(* IEC 61131-3 sources: std_i2980_v2.06_cp053/Source/IMM/ieccontrol/GlobalBaseArchives (part 19) *)

(* ---- ABRegisterDelay.pu ---- *)
(*
@h    ! WARNING !
@h    The Kemro K2 system (including software) only meets category B according to EN 954-1,
@h    thus it is not intended for usage in safety-relevant control applications in the field
@h    of personal safety (e.g. emergency stop).
@h    To implement potentially necessary safety-relevant control tasks, always use additional
@h    external safety devices that are intended for the particular purpose, and meet the necessary
@h    functional safety.
@h    For further information see EN 954-1 (EN ISO 13849-1) and/or the K2-x00 user manual, chapter
@h    "CE conformity, directives and standards".

Delaytime generator for movement and deviceregistration.
*)

ALGORITHM_BLOCK ABRegisterDelay #DUMMY_EDIT_BLOCK

SYSTEM_VAR
 sv_iRegistrationCounter : DINT (* Registrationcounter for delaytime generation *);
END_VAR

(*
Returns a delaytime which is raised by 10ms every call.
*)

ALGORITHM aGet

VAR_OUTPUT
 Time : TIME;
END_VAR
#BEGIN_EDIT_BLOCK
(**************************************** WARNING ********************************************
 *** The KEBA Kemro K2 System including software is not intended for safety control tasks! ***
 ***                       For further information see Comment tab!                        ***
 *********************************************************************************************)

// increment Register counter
sv_iRegistrationCounter := sv_iRegistrationCounter + 1;
// calculate delaytime for registration
Time := T#10ms * sv_iRegistrationCounter;

;#END_EDIT_BLOCK END_ALGORITHM

(*
Resetting the delaytime to make it ready for another registration sequence.
*)

ALGORITHM aReset

#BEGIN_EDIT_BLOCK
(**************************************** WARNING ********************************************
 *** The KEBA Kemro K2 System including software is not intended for safety control tasks! ***
 ***                       For further information see Comment tab!                        ***
 *********************************************************************************************)

// reset devicesRegistered counter
sv_iRegistrationCounter := 0;

;#END_EDIT_BLOCK END_ALGORITHM

END_ALGORITHM_BLOCK

#END_OF_IEC_PART

@Puma @IecEditor 6 10 @Pou 25
@@@BEG_Comment@@@
@h    ! WARNING !
@h    The Kemro K2 system (including software) only meets category B according to EN 954-1,
@h    thus it is not intended for usage in safety-relevant control applications in the field
@h    of personal safety (e.g. emergency stop).
@h    To implement potentially necessary safety-relevant control tasks, always use additional
@h    external safety devices that are intended for the particular purpose, and meet the necessary
@h    functional safety.
@h    For further information see EN 954-1 (EN ISO 13849-1) and/or the K2-x00 user manual, chapter
@h    "CE conformity, directives and standards".

Delaytime generator for movement and deviceregistration.
@@@END_Comment@@@

@BEG_Contents

@BEG_Func
@RT(17)FuncTreeContainer
0
@END_Func

@BEG_Const
@RT(18)ConstTreeContainer
0
@END_Const

@BEG_Export

@BEG_Kind
@ALGORITHM_BLOCK @RT(15)ABRegisterDelay @STRUCTURED_TEXT
@RT(0) @RT(0) @RT(0)
@END_Kind

@BEG_Dcl
@RT(16)DclTreeContainer
1
@Var @RT(23)sv_iRegistrationCounter @RT(0) @T @F @DT @RT(4)DINT @RT(0) @T @T @BASIC 0 @F
@F @F
@T
@BEG_Attrib
3 @RT(0) @RT(44)Registrationcounter for delaytime generation @RT(0)
@END_Attrib
1 8 @F @F @F @F

@END_Dcl

@END_Export

@BEG_Body

2

@BEG_Export

@BEG_Algo
@ALGORITHM @RT(4)aGet @STRUCTURED_TEXT
@RT(0) @RT(0) @RT(0) @F @F
@END_Algo

@BEG_Dcl
@RT(16)DclTreeContainer
1
@Var @RT(4)Time @RT(0) @T @F @DT @RT(4)TIME @RT(0) @T @T @BASIC 0 @F
@F @F
@T
@BEG_Attrib
3 @RT(0) @RT(0) @RT(0)
@END_Attrib
1 3 @F @F @F @F

@END_Dcl

@END_Export

@BEG_Export

@BEG_Algo
@ALGORITHM @RT(6)aReset @STRUCTURED_TEXT
@RT(0) @RT(0) @RT(0) @F @F
@END_Algo

@BEG_Dcl
@RT(16)DclTreeContainer
0
@END_Dcl

@END_Export

@BEG_Body
@TL(10)
(**************************************** WARNING ********************************************
 *** The KEBA Kemro K2 System including software is not intended for safety control tasks! ***
 ***                       For further information see Comment tab!                        ***
 *********************************************************************************************)

// increment Register counter
sv_iRegistrationCounter := sv_iRegistrationCounter + 1;
// calculate delaytime for registration
Time := T#10ms * sv_iRegistrationCounter;

@END_Body

@@@BEG_Comment@@@
@TL(1)
Returns a delaytime which is raised by 10ms every call.
@@@END_Comment@@@

@BEG_Body
@TL(8)
(**************************************** WARNING ********************************************
 *** The KEBA Kemro K2 System including software is not intended for safety control tasks! ***
 ***                       For further information see Comment tab!                        ***
 *********************************************************************************************)

// reset devicesRegistered counter
sv_iRegistrationCounter := 0;

@END_Body

@@@BEG_Comment@@@
@TL(1)
Resetting the delaytime to make it ready for another registration sequence.
@@@END_Comment@@@
@END_Body

@END_Contents

(* ---- ABResourceLockManager.pu ---- *)
IMPORT_OVER_LISTFILE
 STOP_PROCESS_ALGORITHM
, tsResourceLock
, TON

END_IMPORT

ALGORITHM_BLOCK ABResourceLockManager #DUMMY_EDIT_BLOCK

SYSTEM_OBJECT
 PU_Task_7 : TASK;
 TaskSlow : TASK;
END_OBJECT

VAR
 mpResource : REFTO tsResourceLock;
 fbTimeout : TON;
 mbTimeoutUsed : BOOL;
 mName : STRING(31);
END_VAR

ALGORITHM aRequest

#BEGIN_EDIT_BLOCK

IF (mpResource^.iRequest <> 0) THEN // lock request
    IF (mpResource^.iLocked MOD 2 = 0) THEN  // is unlocked
        mpResource^.iResponse := mpResource^.iRequest;
        mpResource^.iLocked := mpResource^.iLocked + 1;  // do lock
        IF (mbTimeoutUsed) THEN
            fbTimeout(IN := FALSE);
            START_PROCESS_ALGORITHM(paTimeout);
        END_IF;
    END_IF;
END_IF;

;#END_EDIT_BLOCK END_ALGORITHM

POSTUPDATE_ALGORITHM pRequest ON PU_Task_7(1) WITH mpResource^.iRequest

#BEGIN_EDIT_BLOCK
aRequest();

;#END_EDIT_BLOCK END_ALGORITHM

POSTUPDATE_ALGORITHM pRelease ON PU_Task_7(2) WITH mpResource^.iResponse

#BEGIN_EDIT_BLOCK
IF (mpResource^.iResponse = 0) THEN
    IF ((mpResource^.iLocked MOD 2 = 1)) THEN // locked
        mpResource^.iLocked := mpResource^.iLocked + 1; // unlock
        mpResource^.iRequest := 0;
        IF (mbTimeoutUsed) THEN
            STOP_PROCESS_ALGORITHM(paTimeout);
        END_IF;
    END_IF;
END_IF;

;#END_EDIT_BLOCK END_ALGORITHM

ALGORITHM aInit

VAR_INPUT
 sName : STRING(31);
 pResource : REFTO tsResourceLock;
 dTimeout : TIME;
END_VAR
#BEGIN_EDIT_BLOCK
mpResource := pResource;
mbTimeoutUsed := dTimeout > T#0s;
fbTimeout.PT := dTimeout;
mName := sName;
aRequest();

;#END_EDIT_BLOCK END_ALGORITHM

PROCESS_ALGORITHM paTimeout ON TaskSlow

VAR
 dummy : DINT;
END_VAR
#BEGIN_EDIT_BLOCK
fbTimeout(IN := (mpResource^.iLocked MOD 2 = 1));
IF (fbTimeout.Q) THEN
    dummy := Print("ABResourceLockManager(%s): lock timeout for lockid 0x%08x", mName, mpResource^.iResponse);
    mpResource^.iResponse := 0;
END_IF;

;#END_EDIT_BLOCK END_ALGORITHM

END_ALGORITHM_BLOCK

#END_OF_IEC_PART

@Puma @IecEditor 6 159 @Pou 25
@@@BEG_Comment@@@

@@@END_Comment@@@

@BEG_Contents

@BEG_Func
@RT(17)FuncTreeContainer
1
@Var @RT(22)STOP_PROCESS_ALGORITHM @RT(0) @T @T @DERIVED 0 @F @RT(23)KEBA_STANDARD_PROCEDURE @F
@T
@BEG_Attrib
0 @RT(0) @RT(0)
@END_Attrib
1 1 @F @F @F @F

@END_Func

@BEG_Const
@RT(18)ConstTreeContainer
0
@END_Const

@BEG_Export

@BEG_Kind
@ALGORITHM_BLOCK @RT(21)ABResourceLockManager @STRUCTURED_TEXT
@RT(0) @RT(0) @RT(0)
@END_Kind

@BEG_Dcl
@RT(16)DclTreeContainer
6
@Var @RT(9)PU_Task_7 @RT(0) @T @T @RENAMED 0 @T @T @DT @RT(4)TASK @RT(0) @T @T @BASIC 0 @F
@F @F
@T
@BEG_Attrib
3 @RT(0) @RT(0) @RT(0)
@END_Attrib
1 7 @F @F @F @F

@Var @RT(10)mpResource @RT(0) @T @T @REFTO 0 @F @DERIVED 0 @T @T @DT @RT(14)tsResourceLock @RT(0) @T @T @UNKNOWN 0 @F
@F @F
@T
@BEG_Attrib
3 @RT(0) @RT(0) @RT(0)
@END_Attrib
1 0 @F @F @F @F

@Var @RT(8)TaskSlow @RT(0) @T @T @RENAMED 0 @T @T @DT @RT(4)TASK @RT(0) @T @T @BASIC 0 @F
@F @F
@T
@BEG_Attrib
3 @RT(0) @RT(0) @RT(0)
@END_Attrib
1 7 @F @F @F @F

@Var @RT(9)fbTimeout @RT(0) @T @T @DERIVED 0 @T @T @DT @RT(3)TON @RT(0) @T @T @UNKNOWN 0 @F
@F @F
@T
@BEG_Attrib
3 @RT(0) @RT(0) @RT(0)
@END_Attrib
1 0 @F @F @F @F

@Var @RT(13)mbTimeoutUsed @RT(0) @T @F @DT @RT(4)BOOL @RT(0) @T @T @BASIC 0 @F
@F @F
@T
@BEG_Attrib
3 @RT(0) @RT(0) @RT(0)
@END_Attrib
1 0 @F @F @F @F

@Var @RT(5)mName @RT(0) @T @F @DT @RT(10)STRING(31) @RT(0) @T @T @STRING 0 @F @RT(2)31 @F
@F @F
@T
@BEG_Attrib
3 @RT(0) @RT(0) @RT(0)
@END_Attrib
1 0 @F @F @F @F

@END_Dcl

@END_Export

@BEG_Body

5

@BEG_Export

@BEG_Algo
@ALGORITHM @RT(8)aRequest @STRUCTURED_TEXT
@RT(0) @RT(0) @RT(0) @F @F
@END_Algo

@BEG_Dcl
@RT(16)DclTreeContainer
0
@END_Dcl

@END_Export

@BEG_Export

@BEG_Algo
@POSTUPDATE_ALGORITHM @RT(8)pRequest @STRUCTURED_TEXT
@RT(0) @RT(20)mpResource^.iRequest @RT(12)PU_Task_7(1) @F @F
@END_Algo

@BEG_Dcl
@RT(16)DclTreeContainer
0
@END_Dcl

@END_Export

@BEG_Export

@BEG_Algo
@POSTUPDATE_ALGORITHM @RT(8)pRelease @STRUCTURED_TEXT
@RT(0) @RT(21)mpResource^.iResponse @RT(12)PU_Task_7(2) @F @F
@END_Algo

@BEG_Dcl
@RT(16)DclTreeContainer
0
@END_Dcl

@END_Export

@BEG_Export

@BEG_Algo
@ALGORITHM @RT(5)aInit @STRUCTURED_TEXT
@RT(0) @RT(0) @RT(0) @F @F
@END_Algo

@BEG_Dcl
@RT(16)DclTreeContainer
3
@Var @RT(5)sName @RT(0) @T @F @DT @RT(10)STRING(31) @RT(0) @T @T @STRING 0 @F @RT(2)31 @F
@F @F
@T
@BEG_Attrib
3 @RT(0) @RT(0) @RT(0)
@END_Attrib
1 1 @F @F @F @F

@Var @RT(9)pResource @RT(0) @T @T @REFTO 0 @F @DERIVED 0 @T @T @DT @RT(14)tsResourceLock @RT(0) @T @T @UNKNOWN 0 @F
@F @F
@T
@BEG_Attrib
3 @RT(0) @RT(0) @RT(0)
@END_Attrib
1 1 @F @F @F @F

@Var @RT(8)dTimeout @RT(0) @T @F @DT @RT(4)TIME @RT(0) @T @T @BASIC 0 @F
@F @F
@T
@BEG_Attrib
3 @RT(0) @RT(0) @RT(0)
@END_Attrib
1 1 @F @F @F @F

@END_Dcl

@END_Export

@BEG_Export

@BEG_Algo
@PROCESS_ALGORITHM @RT(9)paTimeout @STRUCTURED_TEXT
@RT(0) @RT(0) @RT(8)TaskSlow @F @F
@END_Algo

@BEG_Dcl
@RT(16)DclTreeContainer
1
@Var @RT(5)dummy @RT(0) @T @F @DT @RT(4)DINT @RT(0) @T @T @BASIC 0 @F
@F @F
@T
@BEG_Attrib
3 @RT(0) @RT(0) @RT(0)
@END_Attrib
1 0 @F @F @F @F

@END_Dcl

@END_Export

@BEG_Body
@TL(12)

IF (mpResource^.iRequest <> 0) THEN // lock request
    IF (mpResource^.iLocked MOD 2 = 0) THEN  // is unlocked
        mpResource^.iResponse := mpResource^.iRequest;
        mpResource^.iLocked := mpResource^.iLocked + 1;  // do lock
        IF (mbTimeoutUsed) THEN
            fbTimeout(IN := FALSE);
            START_PROCESS_ALGORITHM(paTimeout);
        END_IF;
    END_IF;
END_IF;

@END_Body

@@@BEG_Comment@@@
@TL(0)

@@@END_Comment@@@

@BEG_Body
@TL(2)
aRequest();

@END_Body

@@@BEG_Comment@@@
@TL(0)

@@@END_Comment@@@

@BEG_Body
@TL(10)
IF (mpResource^.iResponse = 0) THEN
    IF ((mpResource^.iLocked MOD 2 = 1)) THEN // locked
        mpResource^.iLocked := mpResource^.iLocked + 1; // unlock
        mpResource^.iRequest := 0;
        IF (mbTimeoutUsed) THEN
            STOP_PROCESS_ALGORITHM(paTimeout);
        END_IF;
    END_IF;
END_IF;

@END_Body

@@@BEG_Comment@@@
@TL(0)

@@@END_Comment@@@

@BEG_Body
@TL(6)
mpResource := pResource;
mbTimeoutUsed := dTimeout > T#0s;
fbTimeout.PT := dTimeout;
mName := sName;
aRequest();

@END_Body

@@@BEG_Comment@@@
@TL(0)

@@@END_Comment@@@

@BEG_Body
@TL(6)
fbTimeout(IN := (mpResource^.iLocked MOD 2 = 1));
IF (fbTimeout.Q) THEN
    dummy := Print("ABResourceLockManager(%s): lock timeout for lockid 0x%08x", mName, mpResource^.iResponse);
    mpResource^.iResponse := 0;
END_IF;

@END_Body

@@@BEG_Comment@@@
@TL(0)

@@@END_Comment@@@
@END_Body

@END_Contents

(* ---- ABStepOutput.pu ---- *)
(*
@h    ! WARNING !
@h    The Kemro K2 system (including software) only meets category B according to EN 954-1,
@h    thus it is not intended for usage in safety-relevant control applications in the field
@h    of personal safety (e.g. emergency stop).
@h    To implement potentially necessary safety-relevant control tasks, always use additional
@h    external safety devices that are intended for the particular purpose, and meet the necessary
@h    functional safety.
@h    For further information see EN 954-1 (EN ISO 13849-1) and/or the K2-x00 user manual, chapter
@h    "CE conformity, directives and standards".

Do step with low and high output value.
*)

IMPORT_OVER_LISTFILE
 GET_TASK_INTERVAL
, cApplPlasticsNoError
, ABConstMovement
, tsVelPre
, tMoveIdent
, R_TRIG

END_IMPORT

ALGORITHM_BLOCK ABStepOutput #DUMMY_EDIT_BLOCK

VAR
 abConstMovement : ABConstMovement;
 CycleTime : TIME (* (of capturing) *);
 bStarted : BOOL;
 mpConstant : REFTO tsVelPre;
 mprMaxSpeed : REFTO REAL;
END_VAR

ALGORITHM aInit

VAR_INPUT
 pConst : REFTO tsVelPre (* pointer to systemvariable that contains profile *);
 MoveId : tMoveIdent (* moveId of constant movement *);
 prMaxSpeed : REFTO REAL;
END_VAR
#BEGIN_EDIT_BLOCK
(**************************************** WARNING ********************************************
 *** The KEBA Kemro K2 System including software is not intended for safety control tasks! ***
 ***                       For further information see Comment tab!                        ***
 *********************************************************************************************)

mpConstant := pConst;

abConstMovement.aInit(pConst := pConst,
                      MoveId := MoveId);

mprMaxSpeed := prMaxSpeed;

;#END_EDIT_BLOCK END_ALGORITHM

(*
Output profile for back pressure calibration
and measure the pressure input
*)

ALGORITHM aRun

VAR_INPUT
 bStart : BOOL (* start constant calib block *);
 bStop : BOOL (* stop constant calib block *);
 bDirection : BOOL (* movement direction *);
 rActPos : REAL (* actual position *);
 rTargetPos : REAL (* target position *);
 bUsePosDetect : BOOL (* TRUE: movement should stop at target position *);
 dDelayTimeOn : TIME (* Delay Time between preoutput and  constoutput *);
 dDelayTimeOff : TIME (* Delay Time between pump stop and bActive FALSE *);
 rPositionUp : REAL;
 rPositionDown : REAL;
 rLowOutput : REAL;
 rHighOutput : REAL;
 dMaxMoveTime : TIME;
 rStopRamp : REAL;
END_VAR

VAR_OUTPUT
 bActive : BOOL (* movement is active *);
 rOutputPre : REAL (* pressure output *);
 rOutputVel : REAL (* velocity output *);
 bPreOutputReached : BOOL (* preoutput ready *);
 bError : BOOL (* flag to indicate if error occured *);
 iErrorInfo : DINT (* additional error info *);
END_VAR

VAR
 fbREdge_Start : R_TRIG;
 iStage : DINT;
 bUeStopRamp : BOOL;
 rSavePreOutput : REAL;
 rSaveRamp : REAL;
 rDownPosition : REAL;
 rUpPosition : REAL;
 dMinDelayTimStop : TIME := T#50ms;
END_VAR
#BEGIN_EDIT_BLOCK
(**************************************** WARNING ********************************************
 *** The KEBA Kemro K2 System including software is not intended for safety control tasks! ***
 ***                       For further information see Comment tab!                        ***
 *********************************************************************************************)

fbREdge_Start(CLK := bStart);
IF fbREdge_Start.Q THEN
   iStage := 1;
   bStarted := TRUE;

   rDownPosition := rPositionDown;
   rUpPosition := rPositionUp;

   rSavePreOutput := mpConstant^.Velocity.PreOutput.rOutputValue;
   mpConstant^.Velocity.PreOutput.rOutputValue :=  rHighOutput;
   mpConstant^.Velocity.PreOutput.rRamp := 1.0e10;
   rSaveRamp := mpConstant^.Velocity.Output.rRamp;

   IF (rStopRamp > 0.0) THEN
      bUeStopRamp := TRUE;
      mpConstant^.Velocity.Output.rRamp := rStopRamp;
   ELSE
      bUeStopRamp := FALSE;
   END_IF;

   abConstMovement.aRun(bStart := FALSE);
   CycleTime := GET_TASK_INTERVAL();
END_IF;
IF bStop THEN
    bStarted := FALSE;
END_IF;

IF bStarted THEN
   //call const movement block
   abConstMovement.aRun(bStart := bStart,
                        bStop := bStop,
                        bDirection := bDirection,
                        rActPos := rActPos,
                        rTargetPos := rTargetPos,
                        bUsePosDetect := bUsePosDetect,
                        rStartOutputPre := 0.0,
                        rStartOutputVel := rHighOutput,
                        dDelayTimeOn := dDelayTimeOn,
                        dDelayTimeOff := MAX(dDelayTimeOff, dMinDelayTimStop),
                        dMaxTime := dMaxMoveTime);

   IF (bDirection AND (rActPos >=  rDownPosition)) OR
      (NOT bDirection AND (rActPos <=  rDownPosition)) THEN
      iStage := 3;
   ELSIF (bDirection AND (rActPos >=  rUpPosition) ) OR
      (NOT bDirection AND (rActPos <=  rUpPosition)) THEN
      iStage := 2;
   END_IF;

   (* to do a jump without a ramp we directly output the low value *)
   IF iStage = 1 THEN
      rOutputVel := MIN(rLowOutput,mpConstant^.Velocity.Output.rOutputValue);
   ELSIF iStage = 2 THEN
      IF (bUeStopRamp) THEN
         rOutputVel := MIN(abConstMovement.aRun.rOutputVel, rHighOutput);
      ELSE
         rOutputVel := rHighOutput;
      END_IF;
   ELSIF iStage = 3 THEN
      IF (bUeStopRamp) THEN
         rOutputVel := abConstMovement.aRun.rOutputVel;
      ELSE
         rOutputVel := MIN(rLowOutput, abConstMovement.aRun.rOutputVel);
      END_IF;
   ELSE
      rOutputVel := 0.0;
   END_IF;

   rOutputPre := abConstMovement.aRun.rOutputPre;
   IF (bDirection AND (rActPos <  rTargetPos)) OR
      (NOT bDirection AND (rActPos >  rTargetPos)) THEN
      bActive := TRUE;
      bPreOutputReached := TRUE;
   ELSE
      bActive := abConstMovement.aRun.bActive;
      bPreOutputReached := abConstMovement.aRun.bPreOutputReached;
   END_IF;

   bError := abConstMovement.aRun.bError;
ELSE
   // not started
   rOutputPre := 0.0;
   rOutputVel := 0.0;
   bPreOutputReached := TRUE;
   bActive := FALSE;
   bError := FALSE;

   abConstMovement.aRun(bStart := FALSE,
                        bStop := TRUE);
END_IF;

//finished ramping down -> switch off
IF bStarted AND NOT abConstMovement.aRun.bActive THEN
   bStarted := FALSE;
   rOutputPre := 0.0;
   rOutputVel := 0.0;
   mpConstant^.Velocity.PreOutput.rOutputValue := rSavePreOutput;
   mpConstant^.Velocity.Output.rRamp := rSaveRamp;
END_IF;

IF abConstMovement.aRun.bError THEN
   mpConstant^.Velocity.PreOutput.rOutputValue := rSavePreOutput;
   mpConstant^.Velocity.Output.rRamp := rSaveRamp;

   IF abConstMovement.aRun.iErrorInfo.Pressure <> cApplPlasticsNoError THEN
      iErrorInfo := abConstMovement.aRun.iErrorInfo.Pressure;
   ELSE
      iErrorInfo := abConstMovement.aRun.iErrorInfo.Velocity;
   END_IF;
   bActive := FALSE;
ELSIF NOT bError THEN
    iErrorInfo := cApplPlasticsNoError;
END_IF;

;#END_EDIT_BLOCK END_ALGORITHM

END_ALGORITHM_BLOCK

#END_OF_IEC_PART

@Puma @IecEditor 6 152 @Pou 25
@@@BEG_Comment@@@
@h    ! WARNING !
@h    The Kemro K2 system (including software) only meets category B according to EN 954-1,
@h    thus it is not intended for usage in safety-relevant control applications in the field
@h    of personal safety (e.g. emergency stop).
@h    To implement potentially necessary safety-relevant control tasks, always use additional
@h    external safety devices that are intended for the particular purpose, and meet the necessary
@h    functional safety.
@h    For further information see EN 954-1 (EN ISO 13849-1) and/or the K2-x00 user manual, chapter
@h    "CE conformity, directives and standards".

Do step with low and high output value.
@@@END_Comment@@@

@BEG_Contents

@BEG_Func
@RT(17)FuncTreeContainer
1
@Var @RT(17)GET_TASK_INTERVAL @RT(0) @T @T @DERIVED 0 @F @RT(22)KEBA_STANDARD_FUNCTION @F
@T
@BEG_Attrib
0 @RT(0) @RT(0)
@END_Attrib
1 1 @F @F @F @F

@END_Func

@BEG_Const
@RT(18)ConstTreeContainer
1
@Var @RT(20)cApplPlasticsNoError @RT(0) @T @F @DT @RT(4)DINT @RT(0) @T @T @BASIC 0 @F
@F @F
@T
@BEG_Attrib
0 @RT(1)0 @RT(8)No Error
@END_Attrib
1 1 @F @F @F @F

@END_Const

@BEG_Export

@BEG_Kind
@ALGORITHM_BLOCK @RT(12)ABStepOutput @STRUCTURED_TEXT
@RT(0) @RT(0) @RT(0)
@END_Kind

@BEG_Dcl
@RT(16)DclTreeContainer
5
@Var @RT(15)abConstMovement @RT(0) @T @T @DERIVED 0 @T @T @DT @RT(15)ABConstMovement @RT(0) @T @T @UNKNOWN 0 @F
@F @F
@T
@BEG_Attrib
3 @RT(0) @RT(0) @RT(0)
@END_Attrib
1 0 @F @F @F @F

@Var @RT(9)CycleTime @RT(0) @T @F @DT @RT(4)TIME @RT(0) @T @T @BASIC 0 @F
@F @F
@T
@BEG_Attrib
3 @RT(0) @RT(14)(of capturing) @RT(0)
@END_Attrib
1 0 @F @F @F @F

@Var @RT(8)bStarted @RT(0) @T @F @DT @RT(4)BOOL @RT(0) @T @T @BASIC 0 @F
@F @F
@T
@BEG_Attrib
3 @RT(0) @RT(0) @RT(0)
@END_Attrib
1 0 @F @F @F @F

@Var @RT(10)mpConstant @RT(0) @T @T @REFTO 0 @F @DERIVED 0 @T @T @DT @RT(8)tsVelPre @RT(0) @T @T @UNKNOWN 0 @F
@F @F
@T
@BEG_Attrib
3 @RT(0) @RT(0) @RT(0)
@END_Attrib
1 0 @F @F @F @F

@Var @RT(11)mprMaxSpeed @RT(0) @T @T @REFTO 0 @T @DT @RT(4)REAL @RT(0) @T @T @BASIC 0 @F
@F @F
@T
@BEG_Attrib
3 @RT(0) @RT(0) @RT(0)
@END_Attrib
1 0 @F @F @F @F

@END_Dcl

@END_Export

@BEG_Body

2

@BEG_Export

@BEG_Algo
@ALGORITHM @RT(5)aInit @STRUCTURED_TEXT
@RT(0) @RT(0) @RT(0) @F @F
@END_Algo

@BEG_Dcl
@RT(16)DclTreeContainer
3
@Var @RT(6)pConst @RT(0) @T @T @REFTO 0 @F @DERIVED 0 @T @T @DT @RT(8)tsVelPre @RT(0) @T @T @UNKNOWN 0 @F
@F @F
@T
@BEG_Attrib
3 @RT(0) @RT(47)pointer to systemvariable that contains profile @RT(0)
@END_Attrib
1 1 @F @F @F @F

@Var @RT(6)MoveId @RT(0) @T @T @DERIVED 0 @T @T @DT @RT(10)tMoveIdent @RT(0) @T @T @UNKNOWN 0 @F
@F @F
@T
@BEG_Attrib
3 @RT(0) @RT(27)moveId of constant movement @RT(0)
@END_Attrib
1 1 @F @F @F @F

@Var @RT(10)prMaxSpeed @RT(0) @T @T @REFTO 0 @T @DT @RT(4)REAL @RT(0) @T @T @BASIC 0 @F
@F @F
@T
@BEG_Attrib
3 @RT(0) @RT(0) @RT(0)
@END_Attrib
1 1 @F @F @F @F

@END_Dcl

@END_Export

@BEG_Export

@BEG_Algo
@ALGORITHM @RT(4)aRun @STRUCTURED_TEXT
@RT(0) @RT(0) @RT(0) @F @F
@END_Algo

@BEG_Dcl
@RT(16)DclTreeContainer
28
@Var @RT(6)bStart @RT(0) @T @F @DT @RT(4)BOOL @RT(0) @T @T @BASIC 0 @F
@F @F
@T
@BEG_Attrib
3 @RT(0) @RT(26)start constant calib block @RT(0)
@END_Attrib
1 1 @F @F @F @F

@Var @RT(5)bStop @RT(0) @T @F @DT @RT(4)BOOL @RT(0) @T @T @BASIC 0 @F
@F @F
@T
@BEG_Attrib
3 @RT(0) @RT(25)stop constant calib block @RT(0)
@END_Attrib
1 1 @F @F @F @F

@Var @RT(10)bDirection @RT(0) @T @F @DT @RT(4)BOOL @RT(0) @T @T @BASIC 0 @F
@F @F
@T
@BEG_Attrib
3 @RT(0) @RT(18)movement direction @RT(0)
@END_Attrib
1 1 @F @F @F @F

@Var @RT(7)rActPos @RT(0) @T @F @DT @RT(4)REAL @RT(0) @T @T @BASIC 0 @F
@F @F
@T
@BEG_Attrib
3 @RT(0) @RT(15)actual position @RT(0)
@END_Attrib
1 1 @F @F @F @F

@Var @RT(10)rTargetPos @RT(0) @T @F @DT @RT(4)REAL @RT(0) @T @T @BASIC 0 @F
@F @F
@T
@BEG_Attrib
3 @RT(0) @RT(15)target position @RT(0)
@END_Attrib
1 1 @F @F @F @F

@Var @RT(13)bUsePosDetect @RT(0) @T @F @DT @RT(4)BOOL @RT(0) @T @T @BASIC 0 @F
@F @F
@T
@BEG_Attrib
3 @RT(0) @RT(45)TRUE: movement should stop at target position @RT(0)
@END_Attrib
1 1 @F @F @F @F

@Var @RT(12)dDelayTimeOn @RT(0) @T @F @DT @RT(4)TIME @RT(0) @T @T @BASIC 0 @F
@F @F
@T
@BEG_Attrib
3 @RT(0) @RT(45)Delay Time between preoutput and  constoutput @RT(0)
@END_Attrib
1 1 @F @F @F @F

@Var @RT(13)dDelayTimeOff @RT(0) @T @F @DT @RT(4)TIME @RT(0) @T @T @BASIC 0 @F
@F @F
@T
@BEG_Attrib
3 @RT(0) @RT(46)Delay Time between pump stop and bActive FALSE @RT(0)
@END_Attrib
1 1 @F @F @F @F

@Var @RT(11)rPositionUp @RT(0) @T @F @DT @RT(4)REAL @RT(0) @T @T @BASIC 0 @F
@F @F
@T
@BEG_Attrib
3 @RT(0) @RT(0) @RT(0)
@END_Attrib
1 1 @F @F @F @F

@Var @RT(13)rPositionDown @RT(0) @T @F @DT @RT(4)REAL @RT(0) @T @T @BASIC 0 @F
@F @F
@T
@BEG_Attrib
3 @RT(0) @RT(0) @RT(0)
@END_Attrib
1 1 @F @F @F @F

@Var @RT(10)rLowOutput @RT(0) @T @F @DT @RT(4)REAL @RT(0) @T @T @BASIC 0 @F
@F @F
@T
@BEG_Attrib
3 @RT(0) @RT(0) @RT(0)
@END_Attrib
1 1 @F @F @F @F

@Var @RT(11)rHighOutput @RT(0) @T @F @DT @RT(4)REAL @RT(0) @T @T @BASIC 0 @F
@F @F
@T
@BEG_Attrib
3 @RT(0) @RT(0) @RT(0)
@END_Attrib
1 1 @F @F @F @F

@Var @RT(12)dMaxMoveTime @RT(0) @T @F @DT @RT(4)TIME @RT(0) @T @T @BASIC 0 @F
@F @F
@T
@BEG_Attrib
3 @RT(0) @RT(0) @RT(0)
@END_Attrib
1 1 @F @F @F @F

@Var @RT(9)rStopRamp @RT(0) @T @F @DT @RT(4)REAL @RT(0) @T @T @BASIC 0 @F
@F @F
@T
@BEG_Attrib
3 @RT(0) @RT(0) @RT(0)
@END_Attrib
1 1 @F @F @F @F

@Var @RT(7)bActive @RT(0) @T @F @DT @RT(4)BOOL @RT(0) @T @T @BASIC 0 @F
@F @F
@T
@BEG_Attrib
3 @RT(0) @RT(18)movement is active @RT(0)
@END_Attrib
1 3 @F @F @F @F

@Var @RT(10)rOutputPre @RT(0) @T @F @DT @RT(4)REAL @RT(0) @T @T @BASIC 0 @F
@F @F
@T
@BEG_Attrib
3 @RT(0) @RT(15)pressure output @RT(0)
@END_Attrib
1 3 @F @F @F @F

@Var @RT(10)rOutputVel @RT(0) @T @F @DT @RT(4)REAL @RT(0) @T @T @BASIC 0 @F
@F @F
@T
@BEG_Attrib
3 @RT(0) @RT(15)velocity output @RT(0)
@END_Attrib
1 3 @F @F @F @F

@Var @RT(17)bPreOutputReached @RT(0) @T @F @DT @RT(4)BOOL @RT(0) @T @T @BASIC 0 @F
@F @F
@T
@BEG_Attrib
3 @RT(0) @RT(15)preoutput ready @RT(0)
@END_Attrib
1 3 @F @F @F @F

@Var @RT(6)bError @RT(0) @T @F @DT @RT(4)BOOL @RT(0) @T @T @BASIC 0 @F
@F @F
@T
@BEG_Attrib
3 @RT(0) @RT(33)flag to indicate if error occured @RT(0)
@END_Attrib
1 3 @F @F @F @F

@Var @RT(10)iErrorInfo @RT(0) @T @F @DT @RT(4)DINT @RT(0) @T @T @BASIC 0 @F
@F @F
@T
@BEG_Attrib
3 @RT(0) @RT(21)additional error info @RT(0)
@END_Attrib
1 3 @F @F @F @F

@Var @RT(13)fbREdge_Start @RT(0) @T @T @DERIVED 0 @T @T @DT @RT(6)R_TRIG @RT(0) @T @T @UNKNOWN 0 @F
@F @F
@T
@BEG_Attrib
3 @RT(0) @RT(0) @RT(0)
@END_Attrib
1 0 @F @F @F @F

@Var @RT(6)iStage @RT(0) @T @F @DT @RT(4)DINT @RT(0) @T @T @BASIC 0 @F
@F @F
@T
@BEG_Attrib
3 @RT(0) @RT(0) @RT(0)
@END_Attrib
1 0 @F @F @F @F

@Var @RT(11)bUeStopRamp @RT(0) @T @F @DT @RT(4)BOOL @RT(0) @T @T @BASIC 0 @F
@F @F
@T
@BEG_Attrib
3 @RT(0) @RT(0) @RT(0)
@END_Attrib
1 0 @F @F @F @F

@Var @RT(14)rSavePreOutput @RT(0) @T @F @DT @RT(4)REAL @RT(0) @T @T @BASIC 0 @F
@F @F
@T
@BEG_Attrib
3 @RT(0) @RT(0) @RT(0)
@END_Attrib
1 0 @F @F @F @F

@Var @RT(9)rSaveRamp @RT(0) @T @F @DT @RT(4)REAL @RT(0) @T @T @BASIC 0 @F
@F @F
@T
@BEG_Attrib
3 @RT(0) @RT(0) @RT(0)
@END_Attrib
1 0 @F @F @F @F

@Var @RT(13)rDownPosition @RT(0) @T @F @DT @RT(4)REAL @RT(0) @T @T @BASIC 0 @F
@F @F
@T
@BEG_Attrib
3 @RT(0) @RT(0) @RT(0)
@END_Attrib
1 0 @F @F @F @F

@Var @RT(11)rUpPosition @RT(0) @T @F @DT @RT(4)REAL @RT(0) @T @T @BASIC 0 @F
@F @F
@T
@BEG_Attrib
3 @RT(0) @RT(0) @RT(0)
@END_Attrib
1 0 @F @F @F @F

@Var @RT(16)dMinDelayTimStop @RT(0) @T @F @DT @RT(4)TIME @RT(0) @T @T @BASIC 0 @F
@F @F
@T
@BEG_Attrib
3 @RT(6)T#50ms @RT(0) @RT(0)
@END_Attrib
1 0 @F @F @F @F

@END_Dcl

@END_Export

@BEG_Body
@TL(13)
(**************************************** WARNING ********************************************
 *** The KEBA Kemro K2 System including software is not intended for safety control tasks! ***
 ***                       For further information see Comment tab!                        ***
 *********************************************************************************************)

mpConstant := pConst;

abConstMovement.aInit(pConst := pConst,
                      MoveId := MoveId);

mprMaxSpeed := prMaxSpeed;

@END_Body

@@@BEG_Comment@@@
@TL(0)

@@@END_Comment@@@

@BEG_Body
@TL(122)
(**************************************** WARNING ********************************************
 *** The KEBA Kemro K2 System including software is not intended for safety control tasks! ***
 ***                       For further information see Comment tab!                        ***
 *********************************************************************************************)

fbREdge_Start(CLK := bStart);
IF fbREdge_Start.Q THEN
   iStage := 1;
   bStarted := TRUE;

   rDownPosition := rPositionDown;
   rUpPosition := rPositionUp;

   rSavePreOutput := mpConstant^.Velocity.PreOutput.rOutputValue;
   mpConstant^.Velocity.PreOutput.rOutputValue :=  rHighOutput;
   mpConstant^.Velocity.PreOutput.rRamp := 1.0e10;
   rSaveRamp := mpConstant^.Velocity.Output.rRamp;

   IF (rStopRamp > 0.0) THEN
      bUeStopRamp := TRUE;
      mpConstant^.Velocity.Output.rRamp := rStopRamp;
   ELSE
      bUeStopRamp := FALSE;
   END_IF;

   abConstMovement.aRun(bStart := FALSE);
   CycleTime := GET_TASK_INTERVAL();
END_IF;
IF bStop THEN
    bStarted := FALSE;
END_IF;

IF bStarted THEN
   //call const movement block
   abConstMovement.aRun(bStart := bStart,
                        bStop := bStop,
                        bDirection := bDirection,
                        rActPos := rActPos,
                        rTargetPos := rTargetPos,
                        bUsePosDetect := bUsePosDetect,
                        rStartOutputPre := 0.0,
                        rStartOutputVel := rHighOutput,
                        dDelayTimeOn := dDelayTimeOn,
                        dDelayTimeOff := MAX(dDelayTimeOff, dMinDelayTimStop),
                        dMaxTime := dMaxMoveTime);

   IF (bDirection AND (rActPos >=  rDownPosition)) OR
      (NOT bDirection AND (rActPos <=  rDownPosition)) THEN
      iStage := 3;
   ELSIF (bDirection AND (rActPos >=  rUpPosition) ) OR
      (NOT bDirection AND (rActPos <=  rUpPosition)) THEN
      iStage := 2;
   END_IF;

   (* to do a jump without a ramp we directly output the low value *)
   IF iStage = 1 THEN
      rOutputVel := MIN(rLowOutput,mpConstant^.Velocity.Output.rOutputValue);
   ELSIF iStage = 2 THEN
      IF (bUeStopRamp) THEN
         rOutputVel := MIN(abConstMovement.aRun.rOutputVel, rHighOutput);
      ELSE
         rOutputVel := rHighOutput;
      END_IF;
   ELSIF iStage = 3 THEN
      IF (bUeStopRamp) THEN
         rOutputVel := abConstMovement.aRun.rOutputVel;
      ELSE
         rOutputVel := MIN(rLowOutput, abConstMovement.aRun.rOutputVel);
      END_IF;
   ELSE
      rOutputVel := 0.0;
   END_IF;

   rOutputPre := abConstMovement.aRun.rOutputPre;
   IF (bDirection AND (rActPos <  rTargetPos)) OR
      (NOT bDirection AND (rActPos >  rTargetPos)) THEN
      bActive := TRUE;
      bPreOutputReached := TRUE;
   ELSE
      bActive := abConstMovement.aRun.bActive;
      bPreOutputReached := abConstMovement.aRun.bPreOutputReached;
   END_IF;

   bError := abConstMovement.aRun.bError;
ELSE
   // not started
   rOutputPre := 0.0;
   rOutputVel := 0.0;
   bPreOutputReached := TRUE;
   bActive := FALSE;
   bError := FALSE;

   abConstMovement.aRun(bStart := FALSE,
                        bStop := TRUE);
END_IF;

//finished ramping down -> switch off
IF bStarted AND NOT abConstMovement.aRun.bActive THEN
   bStarted := FALSE;
   rOutputPre := 0.0;
   rOutputVel := 0.0;
   mpConstant^.Velocity.PreOutput.rOutputValue := rSavePreOutput;
   mpConstant^.Velocity.Output.rRamp := rSaveRamp;
END_IF;

IF abConstMovement.aRun.bError THEN
   mpConstant^.Velocity.PreOutput.rOutputValue := rSavePreOutput;
   mpConstant^.Velocity.Output.rRamp := rSaveRamp;

   IF abConstMovement.aRun.iErrorInfo.Pressure <> cApplPlasticsNoError THEN
      iErrorInfo := abConstMovement.aRun.iErrorInfo.Pressure;
   ELSE
      iErrorInfo := abConstMovement.aRun.iErrorInfo.Velocity;
   END_IF;
   bActive := FALSE;
ELSIF NOT bError THEN
    iErrorInfo := cApplPlasticsNoError;
END_IF;

@END_Body

@@@BEG_Comment@@@
@TL(2)
Output profile for back pressure calibration
and measure the pressure input
@@@END_Comment@@@
@END_Body

@END_Contents

(* ---- ABTargetPosMon.pu ---- *)
(*
@h    ! WARNING !
@h    The Kemro K2 system (including software) only meets category B according to EN 954-1,
@h    thus it is not intended for usage in safety-relevant control applications in the field
@h    of personal safety (e.g. emergency stop).
@h    To implement potentially necessary safety-relevant control tasks, always use additional
@h    external safety devices that are intended for the particular purpose, and meet the necessary
@h    functional safety.
@h    For further information see EN 954-1 (EN ISO 13849-1) and/or the K2-x00 user manual, chapter
@h    "CE conformity, directives and standards".

This AB is used to detect if a target position is reached.
The endposition is reached if actual position is lower or equal / bigger or equal
(depending on the movedirection) than the target position
a given tolerance will also be considered
*)

IMPORT_OVER_LISTFILE
 tsTargetPosData
, KCTRL_LimitSwitch
, KCTRL_LimitSwitch_Param

END_IMPORT

ALGORITHM_BLOCK ABTargetPosMon #DUMMY_EDIT_BLOCK

SYSTEM_VAR
 sv_TargetPosData : tsTargetPosData;
 sv_bInitStart : BOOL;
END_VAR

SYSTEM_OBJECT
 TaskAnalog : TASK;
 PU_Task_3 : TASK;
END_OBJECT

VAR
 abLimitSwitch : KCTRL_LimitSwitch;
 LimitSwitchParam : KCTRL_LimitSwitch_Param;
 mpTolerance : REFTO REAL;
 mprTargetPos : REFTO REAL;
END_VAR

PROCESS_ALGORITHM paRun ON TaskAnalog(3000)

#BEGIN_EDIT_BLOCK
(**************************************** WARNING ********************************************
 *** The KEBA Kemro K2 System including software is not intended for safety control tasks! ***
 ***                       For further information see Comment tab!                        ***
 *********************************************************************************************)

abLimitSwitch.Calculate(rX := sv_TargetPosData.rActPos^);
sv_TargetPosData.pbPosReached^ := abLimitSwitch.Calculate.bY;

;#END_EDIT_BLOCK END_ALGORITHM

POSTUPDATE_ALGORITHM pParameterChanged ON PU_Task_3 WITH mpTolerance^,mprTargetPos^,sv_bInitStart

VAR
 bInitDone : BOOL;
END_VAR
#BEGIN_EDIT_BLOCK
(**************************************** WARNING ********************************************
 *** The KEBA Kemro K2 System including software is not intended for safety control tasks! ***
 ***                       For further information see Comment tab!                        ***
 *********************************************************************************************)

IF NOT bInitDone THEN
    mpTolerance := sv_TargetPosData.rTolerance;
    mprTargetPos := sv_TargetPosData.rTargetPos;
    bInitDone := TRUE;
END_IF;

LimitSwitchParam.rLimit := mprTargetPos^;
LimitSwitchParam.rDiffPEdge := sv_TargetPosData.rTolerance^;
LimitSwitchParam.rDiffNEdge := sv_TargetPosData.rTolerance^;

IF sv_TargetPosData.bDirection THEN
    LimitSwitchParam.bModeInvert := FALSE;
ELSE
    LimitSwitchParam.bModeInvert := TRUE;
END_IF;

abLimitSwitch.Par(Param := LimitSwitchParam);
abLimitSwitch.Init(rX := sv_TargetPosData.rActPos^);

abLimitSwitch.Calculate(rX := sv_TargetPosData.rActPos^);
sv_TargetPosData.pbPosReached^ := abLimitSwitch.Calculate.bY;

START_PROCESS_ALGORITHM(paRun);

;#END_EDIT_BLOCK END_ALGORITHM

END_ALGORITHM_BLOCK

#END_OF_IEC_PART

@Puma @IecEditor 6 22 @Pou 25
@@@BEG_Comment@@@
@h    ! WARNING !
@h    The Kemro K2 system (including software) only meets category B according to EN 954-1,
@h    thus it is not intended for usage in safety-relevant control applications in the field
@h    of personal safety (e.g. emergency stop).
@h    To implement potentially necessary safety-relevant control tasks, always use additional
@h    external safety devices that are intended for the particular purpose, and meet the necessary
@h    functional safety.
@h    For further information see EN 954-1 (EN ISO 13849-1) and/or the K2-x00 user manual, chapter
@h    "CE conformity, directives and standards".

This AB is used to detect if a target position is reached.
The endposition is reached if actual position is lower or equal / bigger or equal
(depending on the movedirection) than the target position
a given tolerance will also be considered
@@@END_Comment@@@

@BEG_Contents

@BEG_Func
@RT(17)FuncTreeContainer
0
@END_Func

@BEG_Const
@RT(18)ConstTreeContainer
0
@END_Const

@BEG_Export

@BEG_Kind
@ALGORITHM_BLOCK @RT(14)ABTargetPosMon @STRUCTURED_TEXT
@RT(0) @RT(0) @RT(0)
@END_Kind

@BEG_Dcl
@RT(16)DclTreeContainer
8
@Var @RT(16)sv_TargetPosData @RT(0) @T @T @DERIVED 0 @T @T @DT @RT(15)tsTargetPosData @RT(0) @T @T @UNKNOWN 0 @F
@F @F
@T
@BEG_Attrib
3 @RT(0) @RT(0) @RT(0)
@END_Attrib
1 8 @F @F @F @F

@Var @RT(10)TaskAnalog @RT(0) @T @T @RENAMED 0 @T @T @DT @RT(4)TASK @RT(0) @T @T @BASIC 0 @F
@F @F
@T
@BEG_Attrib
3 @RT(0) @RT(0) @RT(0)
@END_Attrib
1 7 @F @F @F @F

@Var @RT(13)sv_bInitStart @RT(0) @T @F @DT @RT(4)BOOL @RT(0) @T @T @BASIC 0 @F
@F @F
@T
@BEG_Attrib
3 @RT(0) @RT(0) @RT(0)
@END_Attrib
1 8 @F @F @F @F

@Var @RT(13)abLimitSwitch @RT(0) @T @T @DERIVED 0 @T @T @DT @RT(17)KCTRL_LimitSwitch @RT(0) @T @T @UNKNOWN 0 @F
@F @F
@T
@BEG_Attrib
3 @RT(0) @RT(0) @RT(0)
@END_Attrib
1 0 @F @F @F @F

@Var @RT(16)LimitSwitchParam @RT(0) @T @T @DERIVED 0 @T @T @DT @RT(23)KCTRL_LimitSwitch_Param @RT(0) @T @T @UNKNOWN 0 @F
@F @F
@T
@BEG_Attrib
3 @RT(0) @RT(0) @RT(0)
@END_Attrib
1 0 @F @F @F @F

@Var @RT(11)mpTolerance @RT(0) @T @T @REFTO 0 @T @DT @RT(4)REAL @RT(0) @T @T @BASIC 0 @F
@F @F
@T
@BEG_Attrib
3 @RT(0) @RT(0) @RT(0)
@END_Attrib
1 0 @F @F @F @F

@Var @RT(12)mprTargetPos @RT(0) @T @T @REFTO 0 @T @DT @RT(4)REAL @RT(0) @T @T @BASIC 0 @F
@F @F
@T
@BEG_Attrib
3 @RT(0) @RT(0) @RT(0)
@END_Attrib
1 0 @F @F @F @F

@Var @RT(9)PU_Task_3 @RT(0) @T @T @RENAMED 0 @T @T @DT @RT(4)TASK @RT(0) @T @T @BASIC 0 @F
@F @F
@T
@BEG_Attrib
3 @RT(0) @RT(0) @RT(0)
@END_Attrib
1 7 @F @F @F @F

@END_Dcl

@END_Export

@BEG_Body

2

@BEG_Export

@BEG_Algo
@PROCESS_ALGORITHM @RT(5)paRun @STRUCTURED_TEXT
@RT(0) @RT(0) @RT(16)TaskAnalog(3000) @F @F
@END_Algo

@BEG_Dcl
@RT(16)DclTreeContainer
0
@END_Dcl

@END_Export

@BEG_Export

@BEG_Algo
@POSTUPDATE_ALGORITHM @RT(17)pParameterChanged @STRUCTURED_TEXT
@RT(0) @RT(40)mpTolerance^,mprTargetPos^,sv_bInitStart @RT(9)PU_Task_3 @F @F
@END_Algo

@BEG_Dcl
@RT(16)DclTreeContainer
1
@Var @RT(9)bInitDone @RT(0) @T @F @DT @RT(4)BOOL @RT(0) @T @T @BASIC 0 @F
@F @F
@T
@BEG_Attrib
3 @RT(0) @RT(0) @RT(0)
@END_Attrib
1 0 @F @F @F @F

@END_Dcl

@END_Export

@BEG_Body
@TL(9)
(**************************************** WARNING ********************************************
 *** The KEBA Kemro K2 System including software is not intended for safety control tasks! ***
 ***                       For further information see Comment tab!                        ***
 *********************************************************************************************)

abLimitSwitch.Calculate(rX := sv_TargetPosData.rActPos^);
sv_TargetPosData.pbPosReached^ := abLimitSwitch.Calculate.bY;

@END_Body

@@@BEG_Comment@@@
@TL(0)

@@@END_Comment@@@

@BEG_Body
@TL(30)
(**************************************** WARNING ********************************************
 *** The KEBA Kemro K2 System including software is not intended for safety control tasks! ***
 ***                       For further information see Comment tab!                        ***
 *********************************************************************************************)

IF NOT bInitDone THEN
    mpTolerance := sv_TargetPosData.rTolerance;
    mprTargetPos := sv_TargetPosData.rTargetPos;
    bInitDone := TRUE;
END_IF;

LimitSwitchParam.rLimit := mprTargetPos^;
LimitSwitchParam.rDiffPEdge := sv_TargetPosData.rTolerance^;
LimitSwitchParam.rDiffNEdge := sv_TargetPosData.rTolerance^;

IF sv_TargetPosData.bDirection THEN
    LimitSwitchParam.bModeInvert := FALSE;
ELSE
    LimitSwitchParam.bModeInvert := TRUE;
END_IF;

abLimitSwitch.Par(Param := LimitSwitchParam);
abLimitSwitch.Init(rX := sv_TargetPosData.rActPos^);

abLimitSwitch.Calculate(rX := sv_TargetPosData.rActPos^);
sv_TargetPosData.pbPosReached^ := abLimitSwitch.Calculate.bY;

START_PROCESS_ALGORITHM(paRun);

@END_Body

@@@BEG_Comment@@@
@TL(0)

@@@END_Comment@@@
@END_Body

@END_Contents

(* ---- ABTransducerCalibCycle.pu ---- *)
(*
@h    ! WARNING !
@h    The Kemro K2 system (including software) only meets category B according to EN 954-1,
@h    thus it is not intended for usage in safety-relevant control applications in the field
@h    of personal safety (e.g. emergency stop).
@h    To implement potentially necessary safety-relevant control tasks, always use additional
@h    external safety devices that are intended for the particular purpose, and meet the necessary
@h    functional safety.
@h    For further information see EN 954-1 (EN ISO 13849-1) and/or the K2-x00 user manual, chapter
@h    "CE conformity, directives and standards".

Do automatic transducer calibration with data from sv_TransducerCalibData
move to both ends with outputs specified for setup mode
measuere AI there and write to lintab
*)

IMPORT_OVER_LISTFILE
 SET_ALARM
, SET_EVENT
, CHECK_REF
, tnCalibState_Error
, tnCalibState_Aborted
, tnCalibState_Done
, nSetup
, tnCalibState_Running
, tsCalibMovement
, tnOperationMode
, tsDeviceId
, KCTRL_Lintab_Point
, tsTransducerCalibData
, tevStartRequest
, ABAutoCalibRedoListener
, tyMoveDataArray
, tevStartRequestData
, KAPPL_LintabData_2P
, FBAutoCalibLog
, FBCheckReady
, FBStopStartedMovements
, ABLockList

END_IMPORT

ALGORITHM_BLOCK ABTransducerCalibCycle #DUMMY_EDIT_BLOCK

SYSTEM_VAR
 sv_CalibState : tsCalibMovement;
 sv_OperationMode : tnOperationMode;
 sv_DeviceId : tsDeviceId;
 sv_bDoTransducerCalib : BOOL;
 sv_TmpLintabPoint : KCTRL_Lintab_Point;
 sv_TransducerCalibData : tsTransducerCalibData;
 sv_Movements : tyMoveDataArray;
END_VAR

SYSTEM_OBJECT
 TaskMid : TASK;
 evStartRequest : tevStartRequest;
 PU_Task_7 : TASK;
 erCalibrationStopped : ALARM;
 erCalibrationFailure : ALARM;
 erTransducerCalibNoMovement : ALARM;
 erCalibrationNotActivated : ALARM;
END_OBJECT

VAR
 abAutoCalibRedoListener : ABAutoCalibRedoListener (* not unreferenced used for starting calib *);
END_VAR

PROCESS_ALGORITHM paRun ON TaskMid

VAR_TEMP
 rTmpMax : REAL;
 iCount : DINT;
END_VAR

VAR
 evStartRequestData : tevStartRequestData;
 tmpLintab : KAPPL_LintabData_2P (* temporary lintab for accumulating points *);
 iPos1 : DINT := 1;
 iPos2 : DINT := 2;
 rMinimumVoltageDiff : REAL := 0.7;
 fbLog : FBAutoCalibLog;
 bDoCalibration : BOOL := FALSE;
 bOpenArray : BOOL;
 origLintabPoints : KAPPL_LintabData_2P;
 fbCheckReady : FBCheckReady;
 fbStopStartedMovements : FBStopStartedMovements;
END_VAR

(* IecGraph-Code *)

(* init step *)
INITIAL_STEP S_INIT:
ACheckActivated (P);
END_STEP

ACTION ACheckActivated: #BEGIN_EDIT_BLOCK
bDoCalibration := FALSE;
FOR iCount:=1 TO 20 DO
   IF (sv_Movements[iCount]^.MoveDir = sv_TransducerCalibData.Dir1) AND
      (sv_Movements[iCount]^.MoveId = sv_TransducerCalibData.Id1) THEN
      IF CHECK_REF(sv_Movements[iCount]^.pbActivated) THEN
         IF (sv_Movements[iCount]^.pbActivated^) THEN
            bDoCalibration := TRUE;
         END_IF;
      ELSE
         bDoCalibration := TRUE;
      END_IF;
      EXIT;
   END_IF;
END_FOR;

;#END_EDIT_BLOCK END_ACTION (*ACheckActivated*)

(* steps *)
STEP S_RESET:
AStopmovements (P);
Action24 (P);
END_STEP

ACTION Action24: #BEGIN_EDIT_BLOCK
//restore original transducer-lintab
IF bOpenArray THEN
   sv_CalibState.piUsedLintabPoints^ := origLintabPoints.LintabPoints.uNoOfPoints;
   sv_CalibState.pLintabPoints^[1] := origLintabPoints.LintabPoints.Point[1];
   sv_CalibState.pLintabPoints^[2] := origLintabPoints.LintabPoints.Point[2];
ELSE
   sv_CalibState.pLintab^.LintabPoints.uNoOfPoints := origLintabPoints.LintabPoints.uNoOfPoints;
   sv_CalibState.pLintab^.LintabPoints.Point[1] := origLintabPoints.LintabPoints.Point[1];
   sv_CalibState.pLintab^.LintabPoints.Point[2] := origLintabPoints.LintabPoints.Point[2];
END_IF;

IF sv_CalibState.Status <> tnCalibState_Error THEN
    fbLog('Transducer calib aborted');
    sv_CalibState.Status := tnCalibState_Aborted;
ELSE
    fbLog('Transducer calib error');
END_IF;

;#END_EDIT_BLOCK END_ACTION (*Action24*)
STEP S_STOP:
AStop (P);
END_STEP

ACTION AStop: #BEGIN_EDIT_BLOCK
sv_bDoTransducerCalib := FALSE;
STOP_PROCESS_ALGORITHM();

;#END_EDIT_BLOCK END_ACTION (*AStop*)
STEP S_NOCALIBRATION:
AFinishStep (P);
END_STEP

ACTION AFinishStep: #BEGIN_EDIT_BLOCK
fbLog('Transducer calib not started');
sv_CalibState.Status := tnCalibState_Skipped;
SET_ALARM(Name := erCalibrationNotActivated,
          SubID1 := sv_DeviceId.CompId,
          SubID2 := sv_DeviceId.IndexId);

;#END_EDIT_BLOCK END_ACTION (*AFinishStep*)
STEP Step8:
AInit (P);
END_STEP

STEP S_MOVE1:
AMove1 (P);
ACheckReadyMove1 (N);
END_STEP

ACTION ACheckReadyMove1: #BEGIN_EDIT_BLOCK
fbCheckReady(DeviceId := sv_DeviceId)

;#END_EDIT_BLOCK END_ACTION (*ACheckReadyMove1*)
STEP S_MOVE2:
ASavePos1 (P);
AMove2 (P);
ACheckReadyMove2 (N);
END_STEP

ACTION ASavePos1: #BEGIN_EDIT_BLOCK
fbLog('Transducer direction1 done');
tmpLintab.LintabPoints.Point[iPos2] := sv_TmpLintabPoint;
sv_CalibState.pDisplayLintab^.LintabPoints.Point[iPos2] := sv_TmpLintabPoint;
sv_bDoTransducerCalib := TRUE;

;#END_EDIT_BLOCK END_ACTION (*ASavePos1*)
ACTION ACheckReadyMove2: #BEGIN_EDIT_BLOCK
fbCheckReady(DeviceId := sv_DeviceId);

;#END_EDIT_BLOCK END_ACTION (*ACheckReadyMove2*)
STEP S_CHECK:
ASavePos2 (P);
ACheckSanity (P);
END_STEP

ACTION ASavePos2: #BEGIN_EDIT_BLOCK
fbLog('Transducer direction2 done');
tmpLintab.LintabPoints.Point[iPos1] := sv_TmpLintabPoint;
sv_CalibState.pDisplayLintab^.LintabPoints.Point[iPos1] := sv_TmpLintabPoint;

;#END_EDIT_BLOCK END_ACTION (*ASavePos2*)
ACTION ACheckSanity: #BEGIN_EDIT_BLOCK
// check lintab for sanity, then save it
IF ABS(tmpLintab.LintabPoints.Point[1].rX - tmpLintab.LintabPoints.Point[2].rX) >= rMinimumVoltageDiff AND
   sv_CalibState.Status <> tnCalibState_Error THEN
   IF bOpenArray THEN
      sv_CalibState.piUsedLintabPoints^ := 2;
      sv_CalibState.pLintabPoints^[1] := tmpLintab.LintabPoints.Point[1];
      sv_CalibState.pLintabPoints^[2] := tmpLintab.LintabPoints.Point[2];
   ELSE
      sv_CalibState.pLintab^.LintabPoints.uNoOfPoints := 2;
      sv_CalibState.pLintab^.LintabPoints.Point[1] := tmpLintab.LintabPoints.Point[1];
      sv_CalibState.pLintab^.LintabPoints.Point[2] := tmpLintab.LintabPoints.Point[2];
   END_IF;
   sv_CalibState.Status := tnCalibState_Done;
   fbLog('Transducer finished -> valid');
ELSE
   sv_CalibState.Status := tnCalibState_Error;
   fbLog('Transducer finished -> invalid');
   SET_ALARM(Name := erTransducerCalibNoMovement,
             SubID1 := sv_DeviceId.CompId,
             SubID2 := sv_DeviceId.IndexId);
END_IF;

;#END_EDIT_BLOCK END_ACTION (*ACheckSanity*)

(* transitions *)
GO_ON_TRANSITION Trans15 (* Trans15 *) FROM S_RESET TO S_STOP :=  #BEGIN_EDIT_BLOCK
TRUE
;#END_EDIT_BLOCK
END_TRANSITION

TRANSITION Trans18 (* Trans18 *) FROM S_STOP TO S_INIT :=  #BEGIN_EDIT_BLOCK
TRUE
;#END_EDIT_BLOCK
END_TRANSITION

TRANSITION TStartCalib (* Trans7 *) FROM S_INIT TO Step8 :=  #BEGIN_EDIT_BLOCK
bDoCalibration
;#END_EDIT_BLOCK
END_TRANSITION

TRANSITION TNoCalib (* Trans8 *) FROM S_INIT TO S_NOCALIBRATION :=  #BEGIN_EDIT_BLOCK
NOT bDoCalibration
;#END_EDIT_BLOCK
END_TRANSITION

GO_ON_TRANSITION TCalibStop (* Trans9 *) FROM S_NOCALIBRATION TO S_STOP :=  #BEGIN_EDIT_BLOCK
TRUE
;#END_EDIT_BLOCK
END_TRANSITION

TRANSITION Trans1 (* Trans1 *) FROM Step8 TO S_MOVE1 :=  #BEGIN_EDIT_BLOCK
TRUE
;#END_EDIT_BLOCK
END_TRANSITION

TRANSITION Trans5 (* Trans5 *) FROM S_MOVE1 TO S_MOVE2 :=  #BEGIN_EDIT_BLOCK
fbCheckReady.bReady AND S_MOVE1.T >= t#1s
;#END_EDIT_BLOCK
(*Comment :FIXME: delay because else we sometimes get a erDeviceActive on first movement*)
END_TRANSITION

TRANSITION Trans2 (* Trans2 *) FROM S_MOVE2 TO S_CHECK :=  #BEGIN_EDIT_BLOCK
fbCheckReady.bReady AND S_MOVE2.T >= t#1s
;#END_EDIT_BLOCK
(*Comment :FIXME: delay because else we sometimes get a erDeviceActive on first movement*)
END_TRANSITION

GO_ON_TRANSITION Trans19 (* Trans19 *) FROM S_CHECK TO S_STOP :=  #BEGIN_EDIT_BLOCK
TRUE
;#END_EDIT_BLOCK
END_TRANSITION

(* end IecGraph-Code *)
(* sfc-code *)

(* stand alone actions *)
ACTION AMove1: #BEGIN_EDIT_BLOCK
(**************************************** WARNING ********************************************
 *** The KEBA Kemro K2 System including software is not intended for safety control tasks! ***
 ***                       For further information see Comment tab!                        ***
 *********************************************************************************************)

evStartRequestData.DeviceId := sv_DeviceId;
evStartRequestData.MoveDir := sv_TransducerCalibData.Dir1;
evStartRequestData.MoveId := sv_TransducerCalibData.Id1;
SET_EVENT(evStartRequest, evStartRequestData);

;#END_EDIT_BLOCK END_ACTION (*AMove1*)
ACTION AMove2: #BEGIN_EDIT_BLOCK
(**************************************** WARNING ********************************************
 *** The KEBA Kemro K2 System including software is not intended for safety control tasks! ***
 ***                       For further information see Comment tab!                        ***
 *********************************************************************************************)

evStartRequestData.DeviceId := sv_DeviceId;
evStartRequestData.MoveDir := sv_TransducerCalibData.Dir2;
evStartRequestData.MoveId := sv_TransducerCalibData.Id2;
SET_EVENT(evStartRequest, evStartRequestData);

;#END_EDIT_BLOCK END_ACTION (*AMove2*)
ACTION AStopmovements: #BEGIN_EDIT_BLOCK
(**************************************** WARNING ********************************************
 *** The KEBA Kemro K2 System including software is not intended for safety control tasks! ***
 ***                       For further information see Comment tab!                        ***
 *********************************************************************************************)

fbStopStartedMovements();

;#END_EDIT_BLOCK END_ACTION (*AStopmovements*)
ACTION AInit: #BEGIN_EDIT_BLOCK
(**************************************** WARNING ********************************************
 *** The KEBA Kemro K2 System including software is not intended for safety control tasks! ***
 ***                       For further information see Comment tab!                        ***
 *********************************************************************************************)

// reverse saving of lintab
IF sv_TransducerCalibData.bReverse THEN
    iPos1 := 2;
    iPos2 := 1;
ELSE
    iPos1 := 1;
    iPos2 := 2;
END_IF;
sv_bDoTransducerCalib := TRUE;

//display original lintab
IF CHECK_REF(sv_CalibState.pLintabPoints^) AND CHECK_REF(sv_CalibState.piUsedLintabPoints^) THEN
   bOpenArray := TRUE;
   sv_CalibState.pDisplayLintab^.LintabPoints.Point[1] := sv_CalibState.pLintabPoints^[1];
   sv_CalibState.pDisplayLintab^.LintabPoints.Point[2] := sv_CalibState.pLintabPoints^[2];
ELSE
   bOpenArray := FALSE;
   sv_CalibState.pDisplayLintab^.LintabPoints.Point := sv_CalibState.pLintab^.LintabPoints.Point;
END_IF;
sv_CalibState.pDisplayLintab^.LintabPoints.uNoOfPoints := 2;

// get maximum of transducer
// minimum is always assumed 0
// x is assumed to be Voltage -> 10V
rTmpMax := 0.0;
IF CHECK_REF(sv_TransducerCalibData.prPos1^) THEN
   rTmpMax := sv_TransducerCalibData.prPos1^;
END_IF;
IF CHECK_REF(sv_TransducerCalibData.prPos2^) THEN
   rTmpMax := MAX(rTmpMax, sv_TransducerCalibData.prPos2^);
END_IF;

// change Lintab to [0,0], [10.0, maxStroke] -> avoid erAnalogSensor during calibration
// save data for restoration in case of abortion, error
IF bOpenArray THEN
   origLintabPoints.LintabPoints.uNoOfPoints := sv_CalibState.piUsedLintabPoints^;
   origLintabPoints.LintabPoints.Point[1] := sv_CalibState.pLintabPoints^[1];
   origLintabPoints.LintabPoints.Point[2] := sv_CalibState.pLintabPoints^[2];
   sv_CalibState.piUsedLintabPoints^ := 2;
   sv_CalibState.pLintabPoints^[iPos1].rX := 0.0;
   sv_CalibState.pLintabPoints^[iPos1].rY := 0.0;
   sv_CalibState.pLintabPoints^[iPos2].rX := 10.0;
   sv_CalibState.pLintabPoints^[iPos2].rY := rTmpMax;
ELSE
   origLintabPoints.LintabPoints.uNoOfPoints := sv_CalibState.pLintab^.LintabPoints.uNoOfPoints;
   origLintabPoints.LintabPoints.Point[1] := sv_CalibState.pLintab^.LintabPoints.Point[1];
   origLintabPoints.LintabPoints.Point[2] := sv_CalibState.pLintab^.LintabPoints.Point[2];
   sv_CalibState.pLintab^.LintabPoints.uNoOfPoints := 2;
   sv_CalibState.pLintab^.LintabPoints.Point[iPos1].rX := 0.0;
   sv_CalibState.pLintab^.LintabPoints.Point[iPos1].rY := 0.0;
   sv_CalibState.pLintab^.LintabPoints.Point[iPos2].rX := 10.0;
   sv_CalibState.pLintab^.LintabPoints.Point[iPos2].rY := rTmpMax;
END_IF;

sv_CalibState.prGlobalMaxX^ := 10.0; //V
sv_CalibState.prGlobalMaxY^ := rTmpMax;
fbLog('Transducer calib started');

;#END_EDIT_BLOCK END_ACTION (*AInit*)

(* exits *)

EXIT_TRANSITION E_NotSetupMode := #BEGIN_EDIT_BLOCK
sv_OperationMode <> nSetup
;#END_EDIT_BLOCK
PRIORITY 1 WITH  INITIAL_STEP S_RESET: END_STEP
END_TRANSITION

EXIT_TRANSITION E_NotCalibratingAnymore := #BEGIN_EDIT_BLOCK
// abort calibration, when not in running state and not finished
sv_CalibState.Status <> tnCalibState_Running AND ((*S_INIT.X OR*) S_MOVE1.X OR S_MOVE2.X)
;#END_EDIT_BLOCK
PRIORITY 1 WITH  INITIAL_STEP S_RESET: END_STEP
END_TRANSITION
(* end sfc-code *)

END_ALGORITHM

POSTUPDATE_ALGORITHM pStart ON PU_Task_7 WITH sv_CalibState.Status

VAR
 bLocked : BOOL := FALSE;
 abLockList : ABLockList;
END_VAR
#BEGIN_EDIT_BLOCK
(**************************************** WARNING ********************************************
 *** The KEBA Kemro K2 System including software is not intended for safety control tasks! ***
 ***                       For further information see Comment tab!                        ***
 *********************************************************************************************)

IF sv_OperationMode = nSetup THEN

   IF sv_CalibState.Status = tnCalibState_Running THEN
      // Check if any direction is locked, if it is, calibration start is not meaningful,
      // because it would be stopped later
      bLocked := FALSE;
      abLockList.aCheck(MoveDir:=sv_TransducerCalibData.Dir1, MoveId:=sv_TransducerCalibData.Id1);
      bLocked := abLockList.aCheck.bLocked;
      abLockList.aCheck(MoveDir:=sv_TransducerCalibData.Dir2, MoveId:=sv_TransducerCalibData.Id2);
      bLocked := bLocked OR abLockList.aCheck.bLocked;
      IF bLocked THEN
         sv_CalibState.Status := tnCalibState_Aborted;
         SET_ALARM(erCalibrationStopped);
      ELSE
         START_PROCESS_ALGORITHM(paRun);
      END_IF;
   ELSIF sv_CalibState.Status = tnCalibState_Error THEN
      SET_ALARM(erCalibrationFailure);
   END_IF;

END_IF;

;#END_EDIT_BLOCK END_ALGORITHM

END_ALGORITHM_BLOCK

#END_OF_IEC_PART

@Puma @IecEditor 6 113 @Pou 25
@@@BEG_Comment@@@
@h    ! WARNING !
@h    The Kemro K2 system (including software) only meets category B according to EN 954-1,
@h    thus it is not intended for usage in safety-relevant control applications in the field
@h    of personal safety (e.g. emergency stop).
@h    To implement potentially necessary safety-relevant control tasks, always use additional
@h    external safety devices that are intended for the particular purpose, and meet the necessary
@h    functional safety.
@h    For further information see EN 954-1 (EN ISO 13849-1) and/or the K2-x00 user manual, chapter
@h    "CE conformity, directives and standards".

Do automatic transducer calibration with data from sv_TransducerCalibData
move to both ends with outputs specified for setup mode
measuere AI there and write to lintab
@@@END_Comment@@@

@BEG_Contents

@BEG_Func
@RT(17)FuncTreeContainer
3
@Var @RT(9)SET_ALARM @RT(0) @T @T @DERIVED 0 @F @RT(23)KEBA_STANDARD_PROCEDURE @F
@T
@BEG_Attrib
0 @RT(0) @RT(0)
@END_Attrib
1 1 @F @F @F @F

@Var @RT(9)SET_EVENT @RT(0) @T @T @DERIVED 0 @F @RT(23)KEBA_STANDARD_PROCEDURE @F
@T
@BEG_Attrib
0 @RT(0) @RT(0)
@END_Attrib
1 1 @F @F @F @F

@Var @RT(9)CHECK_REF @RT(0) @T @T @DERIVED 0 @F @RT(23)KEBA_STANDARD_PROCEDURE @F
@T
@BEG_Attrib
0 @RT(0) @RT(0)
@END_Attrib
1 1 @F @F @F @F

@END_Func

@BEG_Const
@RT(18)ConstTreeContainer
5
@Var @RT(18)tnCalibState_Error @RT(0) @T @T @DERIVED 0 @F @RT(12)tnCalibState @F
@T
@BEG_Attrib
0 @RT(1)3 @RT(32)error occured during calibration
@END_Attrib
1 1 @F @F @F @F

@Var @RT(20)tnCalibState_Aborted @RT(0) @T @T @DERIVED 0 @F @RT(12)tnCalibState @F
@T
@BEG_Attrib
0 @RT(1)4 @RT(19)calibration aborted
@END_Attrib
1 1 @F @F @F @F

@Var @RT(17)tnCalibState_Done @RT(0) @T @T @DERIVED 0 @F @RT(12)tnCalibState @F
@T
@BEG_Attrib
0 @RT(1)2 @RT(33)calibration finished successfully
@END_Attrib
1 1 @F @F @F @F

@Var @RT(6)nSetup @RT(0) @T @T @DERIVED 0 @F @RT(15)tnOperationMode @F
@T
@BEG_Attrib
0 @RT(1)0 @RT(36)Setup mode only for service engineer
@END_Attrib
1 1 @F @F @F @F

@Var @RT(20)tnCalibState_Running @RT(0) @T @T @DERIVED 0 @F @RT(12)tnCalibState @F
@T
@BEG_Attrib
0 @RT(1)1 @RT(23)calibration in progress
@END_Attrib
1 1 @F @F @F @F

@END_Const

@BEG_Export

@BEG_Kind
@ALGORITHM_BLOCK @RT(22)ABTransducerCalibCycle @STRUCTURED_TEXT
@RT(0) @RT(0) @RT(0)
@END_Kind

@BEG_Dcl
@RT(16)DclTreeContainer
15
@Var @RT(13)sv_CalibState @RT(0) @T @T @DERIVED 0 @T @T @DT @RT(15)tsCalibMovement @RT(0) @T @T @UNKNOWN 0 @F
@F @F
@T
@BEG_Attrib
3 @RT(0) @RT(0) @RT(0)
@END_Attrib
1 8 @F @F @F @F

@Var @RT(16)sv_OperationMode @RT(0) @T @T @DERIVED 0 @T @T @DT @RT(15)tnOperationMode @RT(0) @T @T @UNKNOWN 0 @F
@F @F
@T
@BEG_Attrib
3 @RT(0) @RT(0) @RT(0)
@END_Attrib
1 8 @F @F @F @F

@Var @RT(11)sv_DeviceId @RT(0) @T @T @DERIVED 0 @T @T @DT @RT(10)tsDeviceId @RT(0) @T @T @UNKNOWN 0 @F
@F @F
@T
@BEG_Attrib
3 @RT(0) @RT(0) @RT(0)
@END_Attrib
1 8 @F @F @F @F

@Var @RT(21)sv_bDoTransducerCalib @RT(0) @T @F @DT @RT(4)BOOL @RT(0) @T @T @BASIC 0 @F
@F @F
@T
@BEG_Attrib
3 @RT(0) @RT(0) @RT(0)
@END_Attrib
1 8 @F @F @F @F

@Var @RT(17)sv_TmpLintabPoint @RT(0) @T @T @DERIVED 0 @T @T @DT @RT(18)KCTRL_Lintab_Point @RT(0) @T @T @UNKNOWN 0 @F
@F @F
@T
@BEG_Attrib
3 @RT(0) @RT(0) @RT(0)
@END_Attrib
1 8 @F @F @F @F

@Var @RT(22)sv_TransducerCalibData @RT(0) @T @T @DERIVED 0 @T @T @DT @RT(21)tsTransducerCalibData @RT(0) @T @T @UNKNOWN 0 @F
@F @F
@T
@BEG_Attrib
3 @RT(0) @RT(0) @RT(0)
@END_Attrib
1 8 @F @F @F @F

@Var @RT(7)TaskMid @RT(0) @T @F @DT @RT(4)TASK @RT(0) @T @T @BASIC 0 @F
@F @F
@T
@BEG_Attrib
3 @RT(0) @RT(0) @RT(0)
@END_Attrib
1 7 @F @F @F @F

@Var @RT(14)evStartRequest @RT(0) @T @T @DERIVED 0 @T @T @DT @RT(15)tevStartRequest @RT(0) @T @T @UNKNOWN 0 @F
@F @F
@T
@BEG_Attrib
3 @RT(0) @RT(0) @RT(0)
@END_Attrib
1 7 @F @F @F @F

@Var @RT(9)PU_Task_7 @RT(0) @T @F @DT @RT(4)TASK @RT(0) @T @T @BASIC 0 @F
@F @F
@T
@BEG_Attrib
3 @RT(0) @RT(0) @RT(0)
@END_Attrib
1 7 @F @F @F @F

@Var @RT(20)erCalibrationStopped @RT(0) @T @F @DT @RT(5)ALARM @RT(0) @T @T @BASIC 0 @F
@F @F
@T
@BEG_Attrib
3 @RT(0) @RT(0) @RT(0)
@END_Attrib
1 7 @F @F @F @F

@Var @RT(20)erCalibrationFailure @RT(0) @T @F @DT @RT(5)ALARM @RT(0) @T @T @BASIC 0 @F
@F @F
@T
@BEG_Attrib
3 @RT(0) @RT(0) @RT(0)
@END_Attrib
1 7 @F @F @F @F

@Var @RT(27)erTransducerCalibNoMovement @RT(0) @T @F @DT @RT(5)ALARM @RT(0) @T @T @BASIC 0 @F
@F @F
@T
@BEG_Attrib
3 @RT(0) @RT(0) @RT(0)
@END_Attrib
1 7 @F @F @F @F

@Var @RT(23)abAutoCalibRedoListener @RT(0) @T @T @DERIVED 0 @T @T @DT @RT(23)ABAutoCalibRedoListener @RT(0) @T @T @UNKNOWN 0 @F
@F @F
@T
@BEG_Attrib
3 @RT(0) @RT(40)not unreferenced used for starting calib @RT(0)
@END_Attrib
1 0 @F @F @F @F

@Var @RT(12)sv_Movements @RT(0) @T @T @DERIVED 0 @T @T @DT @RT(15)tyMoveDataArray @RT(0) @T @T @UNKNOWN 0 @F
@F @F
@T
@BEG_Attrib
3 @RT(0) @RT(0) @RT(0)
@END_Attrib
1 8 @F @F @F @F

@Var @RT(25)erCalibrationNotActivated @RT(0) @T @F @DT @RT(5)ALARM @RT(0) @T @T @BASIC 0 @F
@F @F
@T
@BEG_Attrib
3 @RT(0) @RT(0) @RT(0)
@END_Attrib
1 7 @F @F @F @F

@END_Dcl

@END_Export

@BEG_Body

2

@BEG_Export

@BEG_Algo
@PROCESS_ALGORITHM @RT(5)paRun @SEQUENTIAL_FLOW_CHART
@RT(0) @RT(0) @RT(7)TaskMid @F @F
@END_Algo

@BEG_Dcl
@RT(16)DclTreeContainer
13
@Var @RT(7)rTmpMax @RT(0) @T @F @DT @RT(4)REAL @RT(0) @T @T @BASIC 0 @F
@F @F
@T
@BEG_Attrib
3 @RT(0) @RT(0) @RT(0)
@END_Attrib
1 4 @F @F @F @F

@Var @RT(18)evStartRequestData @RT(0) @T @T @DERIVED 0 @T @T @DT @RT(19)tevStartRequestData @RT(0) @T @T @UNKNOWN 0 @F
@F @F
@T
@BEG_Attrib
3 @RT(0) @RT(0) @RT(0)
@END_Attrib
1 0 @F @F @F @F

@Var @RT(9)tmpLintab @RT(0) @T @T @DERIVED 0 @T @T @DT @RT(19)KAPPL_LintabData_2P @RT(0) @T @T @UNKNOWN 0 @F
@F @F
@T
@BEG_Attrib
3 @RT(0) @RT(40)temporary lintab for accumulating points @RT(0)
@END_Attrib
1 0 @F @F @F @F

@Var @RT(5)iPos1 @RT(0) @T @F @DT @RT(4)DINT @RT(0) @T @T @BASIC 0 @F
@F @F
@T
@BEG_Attrib
3 @RT(1)1 @RT(0) @RT(0)
@END_Attrib
1 0 @F @F @F @F

@Var @RT(5)iPos2 @RT(0) @T @F @DT @RT(4)DINT @RT(0) @T @T @BASIC 0 @F
@F @F
@T
@BEG_Attrib
3 @RT(1)2 @RT(0) @RT(0)
@END_Attrib
1 0 @F @F @F @F

@Var @RT(19)rMinimumVoltageDiff @RT(0) @T @F @DT @RT(4)REAL @RT(0) @T @T @BASIC 0 @F
@F @F
@T
@BEG_Attrib
3 @RT(3)0.7 @RT(0) @RT(0)
@END_Attrib
1 0 @F @F @F @F

@Var @RT(5)fbLog @RT(0) @T @T @DERIVED 0 @T @T @DT @RT(14)FBAutoCalibLog @RT(0) @T @T @UNKNOWN 0 @F
@F @F
@T
@BEG_Attrib
3 @RT(0) @RT(0) @RT(0)
@END_Attrib
1 0 @F @F @F @F

@Var @RT(14)bDoCalibration @RT(0) @T @F @DT @RT(4)BOOL @RT(0) @T @T @BASIC 0 @F
@F @F
@T
@BEG_Attrib
3 @RT(5)FALSE @RT(0) @RT(0)
@END_Attrib
1 0 @F @F @F @F

@Var @RT(6)iCount @RT(0) @T @F @DT @RT(4)DINT @RT(0) @T @T @BASIC 0 @F
@F @F
@T
@BEG_Attrib
3 @RT(0) @RT(0) @RT(0)
@END_Attrib
1 4 @F @F @F @F

@Var @RT(10)bOpenArray @RT(0) @T @F @DT @RT(4)BOOL @RT(0) @T @T @BASIC 0 @F
@F @F
@T
@BEG_Attrib
3 @RT(0) @RT(0) @RT(0)
@END_Attrib
1 0 @F @F @F @F

@Var @RT(16)origLintabPoints @RT(0) @T @T @DERIVED 0 @T @T @DT @RT(19)KAPPL_LintabData_2P @RT(0) @T @T @UNKNOWN 0 @F
@F @F
@T
@BEG_Attrib
3 @RT(0) @RT(0) @RT(0)
@END_Attrib
1 0 @F @F @F @F

@Var @RT(12)fbCheckReady @RT(0) @T @T @DERIVED 0 @T @T @DT @RT(12)FBCheckReady @RT(0) @T @T @UNKNOWN 0 @F
@F @F
@T
@BEG_Attrib
3 @RT(0) @RT(0) @RT(0)
@END_Attrib
1 0 @F @F @F @F

@Var @RT(22)fbStopStartedMovements @RT(0) @T @T @DERIVED 0 @T @T @DT @RT(22)FBStopStartedMovements @RT(0) @T @T @UNKNOWN 0 @F
@F @F
@T
@BEG_Attrib
3 @RT(0) @RT(0) @RT(0)
@END_Attrib
1 0 @F @F @F @F

@END_Dcl

@END_Export

@BEG_Export

@BEG_Algo
@POSTUPDATE_ALGORITHM @RT(6)pStart @STRUCTURED_TEXT
@RT(0) @RT(20)sv_CalibState.Status @RT(9)PU_Task_7 @F @F
@END_Algo

@BEG_Dcl
@RT(16)DclTreeContainer
2
@Var @RT(7)bLocked @RT(0) @T @F @DT @RT(4)BOOL @RT(0) @T @T @BASIC 0 @F
@F @F
@T
@BEG_Attrib
3 @RT(5)FALSE @RT(0) @RT(0)
@END_Attrib
1 0 @F @F @F @F

@Var @RT(10)abLockList @RT(0) @T @T @DERIVED 0 @T @T @DT @RT(10)ABLockList @RT(0) @T @T @UNKNOWN 0 @F
@F @F
@T
@BEG_Attrib
3 @RT(0) @RT(0) @RT(0)
@END_Attrib
1 0 @F @F @F @F

@END_Dcl

@END_Export

@BEG_SfcBody
16 10 10

@BEG_SfcData 2
@StepSeq @RT(4)sseq @F 15
@Step @RT(7)S_RESET @F @F @T @F @RT(0) @F
@AcbCont @RT(7)unnamed @F 2
@Acb @RT(14)AStopmovements @F @F @RT(1)P @RT(0) @F @F @F @F
@Acb @RT(8)Action24 @F @T @RT(1)P @RT(0) @F @F @T @TL(18)
//restore original transducer-lintab
IF bOpenArray THEN
   sv_CalibState.piUsedLintabPoints^ := origLintabPoints.LintabPoints.uNoOfPoints;
   sv_CalibState.pLintabPoints^[1] := origLintabPoints.LintabPoints.Point[1];
   sv_CalibState.pLintabPoints^[2] := origLintabPoints.LintabPoints.Point[2];
ELSE
   sv_CalibState.pLintab^.LintabPoints.uNoOfPoints := origLintabPoints.LintabPoints.uNoOfPoints;
   sv_CalibState.pLintab^.LintabPoints.Point[1] := origLintabPoints.LintabPoints.Point[1];
   sv_CalibState.pLintab^.LintabPoints.Point[2] := origLintabPoints.LintabPoints.Point[2];
END_IF;

IF sv_CalibState.Status <> tnCalibState_Error THEN
    fbLog('Transducer calib aborted');
    sv_CalibState.Status := tnCalibState_Aborted;
ELSE
    fbLog('Transducer calib error');
END_IF;

@F

@Trans @RT(7)Trans15 @F @T @F @F @T @F @TL(2)
TRUE

@RT(7)Trans15 @F
@Step @RT(6)S_STOP @F @F @T @F @RT(0) @F
@AcbCont @RT(7)unnamed @F 1
@Acb @RT(5)AStop @F @T @RT(1)P @RT(0) @F @F @T @TL(3)
sv_bDoTransducerCalib := FALSE;
STOP_PROCESS_ALGORITHM();

@F

@Trans @RT(7)Trans18 @F @T @F @F @T @T @TL(2)
TRUE

@RT(7)Trans18 @F
@Step @RT(6)S_INIT @F @T @F @F @RT(0) @F
@AcbCont @RT(7)unnamed @F 1
@Acb @RT(15)ACheckActivated @F @T @RT(1)P @RT(0) @F @F @T @TL(15)
bDoCalibration := FALSE;
FOR iCount:=1 TO 20 DO
   IF (sv_Movements[iCount]^.MoveDir = sv_TransducerCalibData.Dir1) AND
      (sv_Movements[iCount]^.MoveId = sv_TransducerCalibData.Id1) THEN
      IF CHECK_REF(sv_Movements[iCount]^.pbActivated) THEN
         IF (sv_Movements[iCount]^.pbActivated^) THEN
            bDoCalibration := TRUE;
         END_IF;
      ELSE
         bDoCalibration := TRUE;
      END_IF;
      EXIT;
   END_IF;
END_FOR;

@F

@AltBranch @RT(3)alt @F 2
@TransSeq @RT(4)tseq @F 1
@Trans @RT(11)TStartCalib @F @T @F @F @T @T @TL(2)
bDoCalibration

@RT(6)Trans7 @F

@TransSeq @RT(4)tseq @F 4
@Trans @RT(8)TNoCalib @F @T @F @F @T @T @TL(2)
NOT bDoCalibration

@RT(6)Trans8 @F
@Step @RT(15)S_NOCALIBRATION @F @F @F @F @RT(0) @F
@AcbCont @RT(7)unnamed @F 1
@Acb @RT(11)AFinishStep @F @T @RT(1)P @RT(0) @F @F @T @TL(6)
fbLog('Transducer calib not started');
sv_CalibState.Status := tnCalibState_Skipped;
SET_ALARM(Name := erCalibrationNotActivated,
          SubID1 := sv_DeviceId.CompId,
          SubID2 := sv_DeviceId.IndexId);

@F

@Trans @RT(10)TCalibStop @F @T @F @F @T @F @TL(2)
TRUE

@RT(6)Trans9 @F
@Goto @RT(6)S_STOP @F @F

@Step @RT(5)Step8 @F @F @F @F @RT(0) @F
@AcbCont @RT(7)unnamed @F 1
@Acb @RT(5)AInit @F @F @RT(1)P @RT(0) @F @F @F @F

@Trans @RT(6)Trans1 @F @T @F @F @T @T @TL(2)
TRUE

@RT(6)Trans1 @F
@Step @RT(7)S_MOVE1 @F @F @F @F @RT(0) @F
@AcbCont @RT(7)unnamed @F 2
@Acb @RT(6)AMove1 @F @F @RT(1)P @RT(0) @F @F @F @F
@Acb @RT(16)ACheckReadyMove1 @F @T @RT(1)N @RT(0) @F @F @T @TL(2)
fbCheckReady(DeviceId := sv_DeviceId)

@F

@Trans @RT(6)Trans5 @F @T @F @F @T @T @TL(2)
fbCheckReady.bReady AND S_MOVE1.T >= t#1s

@RT(6)Trans5 @T @TL(1)
Comment :FIXME: delay because else we sometimes get a erDeviceActive on first movement

@Step @RT(7)S_MOVE2 @F @F @F @F @RT(0) @F
@AcbCont @RT(7)unnamed @F 3
@Acb @RT(9)ASavePos1 @F @T @RT(1)P @RT(0) @F @F @T @TL(5)
fbLog('Transducer direction1 done');
tmpLintab.LintabPoints.Point[iPos2] := sv_TmpLintabPoint;
sv_CalibState.pDisplayLintab^.LintabPoints.Point[iPos2] := sv_TmpLintabPoint;
sv_bDoTransducerCalib := TRUE;

@F
@Acb @RT(6)AMove2 @F @F @RT(1)P @RT(0) @F @F @F @F
@Acb @RT(16)ACheckReadyMove2 @F @T @RT(1)N @RT(0) @F @F @T @TL(2)
fbCheckReady(DeviceId := sv_DeviceId);

@F

@Trans @RT(6)Trans2 @F @T @F @F @T @T @TL(2)
fbCheckReady.bReady AND S_MOVE2.T >= t#1s

@RT(6)Trans2 @T @TL(1)
Comment :FIXME: delay because else we sometimes get a erDeviceActive on first movement

@Step @RT(7)S_CHECK @F @F @F @F @RT(0) @F
@AcbCont @RT(7)unnamed @F 2
@Acb @RT(9)ASavePos2 @F @T @RT(1)P @RT(0) @F @F @T @TL(4)
fbLog('Transducer direction2 done');
tmpLintab.LintabPoints.Point[iPos1] := sv_TmpLintabPoint;
sv_CalibState.pDisplayLintab^.LintabPoints.Point[iPos1] := sv_TmpLintabPoint;

@F
@Acb @RT(12)ACheckSanity @F @T @RT(1)P @RT(0) @F @F @T @TL(22)
// check lintab for sanity, then save it
IF ABS(tmpLintab.LintabPoints.Point[1].rX - tmpLintab.LintabPoints.Point[2].rX) >= rMinimumVoltageDiff AND
   sv_CalibState.Status <> tnCalibState_Error THEN
   IF bOpenArray THEN
      sv_CalibState.piUsedLintabPoints^ := 2;
      sv_CalibState.pLintabPoints^[1] := tmpLintab.LintabPoints.Point[1];
      sv_CalibState.pLintabPoints^[2] := tmpLintab.LintabPoints.Point[2];
   ELSE
      sv_CalibState.pLintab^.LintabPoints.uNoOfPoints := 2;
      sv_CalibState.pLintab^.LintabPoints.Point[1] := tmpLintab.LintabPoints.Point[1];
      sv_CalibState.pLintab^.LintabPoints.Point[2] := tmpLintab.LintabPoints.Point[2];
   END_IF;
   sv_CalibState.Status := tnCalibState_Done;
   fbLog('Transducer finished -> valid');
ELSE
   sv_CalibState.Status := tnCalibState_Error;
   fbLog('Transducer finished -> invalid');
   SET_ALARM(Name := erTransducerCalibNoMovement,
             SubID1 := sv_DeviceId.CompId,
             SubID2 := sv_DeviceId.IndexId);
END_IF;

@F

@Trans @RT(7)Trans19 @F @T @F @F @T @F @TL(2)
TRUE

@RT(7)Trans19 @F
@Goto @RT(6)S_STOP @F @F
@END_SfcData
@SaActions 4
@SaText @RT(6)AMove1 1 @TL(10)
(**************************************** WARNING ********************************************
 *** The KEBA Kemro K2 System including software is not intended for safety control tasks! ***
 ***                       For further information see Comment tab!                        ***
 *********************************************************************************************)

evStartRequestData.DeviceId := sv_DeviceId;
evStartRequestData.MoveDir := sv_TransducerCalibData.Dir1;
evStartRequestData.MoveId := sv_TransducerCalibData.Id1;
SET_EVENT(evStartRequest, evStartRequestData);

@SaText @RT(6)AMove2 1 @TL(10)
(**************************************** WARNING ********************************************
 *** The KEBA Kemro K2 System including software is not intended for safety control tasks! ***
 ***                       For further information see Comment tab!                        ***
 *********************************************************************************************)

evStartRequestData.DeviceId := sv_DeviceId;
evStartRequestData.MoveDir := sv_TransducerCalibData.Dir2;
evStartRequestData.MoveId := sv_TransducerCalibData.Id2;
SET_EVENT(evStartRequest, evStartRequestData);

@SaText @RT(14)AStopmovements 1 @TL(7)
(**************************************** WARNING ********************************************
 *** The KEBA Kemro K2 System including software is not intended for safety control tasks! ***
 ***                       For further information see Comment tab!                        ***
 *********************************************************************************************)

fbStopStartedMovements();

@SaText @RT(5)AInit 1 @TL(63)
(**************************************** WARNING ********************************************
 *** The KEBA Kemro K2 System including software is not intended for safety control tasks! ***
 ***                       For further information see Comment tab!                        ***
 *********************************************************************************************)

// reverse saving of lintab
IF sv_TransducerCalibData.bReverse THEN
    iPos1 := 2;
    iPos2 := 1;
ELSE
    iPos1 := 1;
    iPos2 := 2;
END_IF;
sv_bDoTransducerCalib := TRUE;

//display original lintab
IF CHECK_REF(sv_CalibState.pLintabPoints^) AND CHECK_REF(sv_CalibState.piUsedLintabPoints^) THEN
   bOpenArray := TRUE;
   sv_CalibState.pDisplayLintab^.LintabPoints.Point[1] := sv_CalibState.pLintabPoints^[1];
   sv_CalibState.pDisplayLintab^.LintabPoints.Point[2] := sv_CalibState.pLintabPoints^[2];
ELSE
   bOpenArray := FALSE;
   sv_CalibState.pDisplayLintab^.LintabPoints.Point := sv_CalibState.pLintab^.LintabPoints.Point;
END_IF;
sv_CalibState.pDisplayLintab^.LintabPoints.uNoOfPoints := 2;

// get maximum of transducer
// minimum is always assumed 0
// x is assumed to be Voltage -> 10V
rTmpMax := 0.0;
IF CHECK_REF(sv_TransducerCalibData.prPos1^) THEN
   rTmpMax := sv_TransducerCalibData.prPos1^;
END_IF;
IF CHECK_REF(sv_TransducerCalibData.prPos2^) THEN
   rTmpMax := MAX(rTmpMax, sv_TransducerCalibData.prPos2^);
END_IF;

// change Lintab to [0,0], [10.0, maxStroke] -> avoid erAnalogSensor during calibration
// save data for restoration in case of abortion, error
IF bOpenArray THEN
   origLintabPoints.LintabPoints.uNoOfPoints := sv_CalibState.piUsedLintabPoints^;
   origLintabPoints.LintabPoints.Point[1] := sv_CalibState.pLintabPoints^[1];
   origLintabPoints.LintabPoints.Point[2] := sv_CalibState.pLintabPoints^[2];
   sv_CalibState.piUsedLintabPoints^ := 2;
   sv_CalibState.pLintabPoints^[iPos1].rX := 0.0;
   sv_CalibState.pLintabPoints^[iPos1].rY := 0.0;
   sv_CalibState.pLintabPoints^[iPos2].rX := 10.0;
   sv_CalibState.pLintabPoints^[iPos2].rY := rTmpMax;
ELSE
   origLintabPoints.LintabPoints.uNoOfPoints := sv_CalibState.pLintab^.LintabPoints.uNoOfPoints;
   origLintabPoints.LintabPoints.Point[1] := sv_CalibState.pLintab^.LintabPoints.Point[1];
   origLintabPoints.LintabPoints.Point[2] := sv_CalibState.pLintab^.LintabPoints.Point[2];
   sv_CalibState.pLintab^.LintabPoints.uNoOfPoints := 2;
   sv_CalibState.pLintab^.LintabPoints.Point[iPos1].rX := 0.0;
   sv_CalibState.pLintab^.LintabPoints.Point[iPos1].rY := 0.0;
   sv_CalibState.pLintab^.LintabPoints.Point[iPos2].rX := 10.0;
   sv_CalibState.pLintab^.LintabPoints.Point[iPos2].rY := rTmpMax;
END_IF;

sv_CalibState.prGlobalMaxX^ := 10.0; //V
sv_CalibState.prGlobalMaxY^ := rTmpMax;
fbLog('Transducer calib started');

@SaTrans 0
@SaExits 2
@SaExit @SaText @RT(14)E_NotSetupMode 1 @TL(2)
sv_OperationMode <> nSetup

@RT(7)S_RESET @RT(1)1 @F @F @SaSfc @RT(14)E_NotSetupMode 5 @RT(5)DUMMY
@BEG_SfcData 2
@ExitSeq @RT(4)sseq @F 3
@Step @RT(8)unnamed1 @F @T @F @F @RT(0) @F
@AcbCont @RT(7)unnamed @F 0

@Trans @RT(8)unnamed3 @F @T @F @F @T @T @TL(2)

@RT(8)unnamed3 @F
@Goto @RT(9)unlabeled @F @F
@END_SfcData

@SaExit @SaText @RT(23)E_NotCalibratingAnymore 1 @TL(3)
// abort calibration, when not in running state and not finished
sv_CalibState.Status <> tnCalibState_Running AND ((*S_INIT.X OR*) S_MOVE1.X OR S_MOVE2.X)

@RT(7)S_RESET @RT(1)1 @F @F @SaSfc @RT(23)E_NotCalibratingAnymore 5 @RT(5)DUMMY
@BEG_SfcData 2
@ExitSeq @RT(4)sseq @F 3
@Step @RT(8)unnamed4 @F @T @F @F @RT(0) @F
@AcbCont @RT(7)unnamed @F 0

@Trans @RT(8)unnamed6 @F @T @F @F @T @T @TL(2)

@RT(8)unnamed6 @F
@Goto @RT(9)unlabeled @F @F
@END_SfcData

@END_SfcBody

@@@BEG_Comment@@@
@TL(0)

@@@END_Comment@@@

@BEG_Body
@TL(28)
(**************************************** WARNING ********************************************
 *** The KEBA Kemro K2 System including software is not intended for safety control tasks! ***
 ***                       For further information see Comment tab!                        ***
 *********************************************************************************************)

IF sv_OperationMode = nSetup THEN

   IF sv_CalibState.Status = tnCalibState_Running THEN
      // Check if any direction is locked, if it is, calibration start is not meaningful,
      // because it would be stopped later
      bLocked := FALSE;
      abLockList.aCheck(MoveDir:=sv_TransducerCalibData.Dir1, MoveId:=sv_TransducerCalibData.Id1);
      bLocked := abLockList.aCheck.bLocked;
      abLockList.aCheck(MoveDir:=sv_TransducerCalibData.Dir2, MoveId:=sv_TransducerCalibData.Id2);
      bLocked := bLocked OR abLockList.aCheck.bLocked;
      IF bLocked THEN
         sv_CalibState.Status := tnCalibState_Aborted;
         SET_ALARM(erCalibrationStopped);
      ELSE
         START_PROCESS_ALGORITHM(paRun);
      END_IF;
   ELSIF sv_CalibState.Status = tnCalibState_Error THEN
      SET_ALARM(erCalibrationFailure);
   END_IF;

END_IF;

@END_Body

@@@BEG_Comment@@@
@TL(0)

@@@END_Comment@@@
@END_Body

@END_Contents

(* ---- ABUpdateRelLintabPre.pu ---- *)
(*
@h    ! WARNING !
@h    The Kemro K2 system (including software) only meets category B according to EN 954-1,
@h    thus it is not intended for usage in safety-relevant control applications in the field
@h    of personal safety (e.g. emergency stop).
@h    To implement potentially necessary safety-relevant control tasks, always use additional
@h    external safety devices that are intended for the particular purpose, and meet the necessary
@h    functional safety.
@h    For further information see EN 954-1 (EN ISO 13849-1) and/or the K2-x00 user manual, chapter
@h    "CE conformity, directives and standards".
*)

IMPORT_OVER_LISTFILE
 FFixCylinderData
, FCalculateCylinderSize
, CHECK_REF
, KAPPL_LintabData
, tsCylinderData
, FBDebugTrace

END_IMPORT

ALGORITHM_BLOCK ABUpdateRelLintabPre #DUMMY_EDIT_BLOCK

SYSTEM_VAR
 sv_bCalcMaxValuesFromCylData : BOOL (* TRUE: calculate max speed and max pressure values by using cylinder data;  FALSE: max values must be entered manually *);
END_VAR

SYSTEM_OBJECT
 PU_Task_7 : TASK;
END_OBJECT

VAR
 mpLintabOut : REFTO KAPPL_LintabData (* refto pressure lintab of movement *);
 mpCylinderData : REFTO tsCylinderData (* refto cylinder data *);
 mprMaxPressure : REFTO REAL (* reference to calculated max. pressure of movement *);
 mprMaxHydrPressure : REFTO REAL (* reference to max. hydraulic pressure *);
 mbInitDone : BOOL;
 mbUseForce : BOOL;
 mbFwd : BOOL;
END_VAR

ALGORITHM aUpdateLintabOut

#BEGIN_EDIT_BLOCK
(**************************************** WARNING ********************************************
 *** The KEBA Kemro K2 System including software is not intended for safety control tasks! ***
 ***                       For further information see Comment tab!                        ***
 *********************************************************************************************)

// save data to Pre lintab
// normally a 1:1 lintab
mpLintabOut^.LintabPoints.uNoOfPoints := 2;
mpLintabOut^.LintabPoints.Point[1].rX := 0.0;
mpLintabOut^.LintabPoints.Point[1].rY := 0.0;
mpLintabOut^.LintabPoints.Point[2].rX := mprMaxPressure^;
mpLintabOut^.LintabPoints.Point[2].rY := mprMaxHydrPressure^;

;#END_EDIT_BLOCK END_ALGORITHM

ALGORITHM aCalcMaxPressure

VAR_TEMP
 rCylinderSize : REAL (* size of cylinder im mm˛ *);
 tmp : BOOL;
END_VAR

VAR
 bSmallSize : BOOL;
END_VAR
#BEGIN_EDIT_BLOCK
(**************************************** WARNING ********************************************
 *** The KEBA Kemro K2 System including software is not intended for safety control tasks! ***
 ***                       For further information see Comment tab!                        ***
 *********************************************************************************************)

IF NOT sv_bCalcMaxValuesFromCylData THEN
   // no calculation necessary
   RETURN;
END_IF;

IF mbUseForce THEN
   tmp := FFixCylinderData(mpCylinderData);
   bSmallSize := mbFwd AND mpCylinderData^.bUseSmallSize OR
                 ((NOT mbFwd AND NOT mpCylinderData^.bUseSmallSize));
   rCylinderSize := FCalculateCylinderSize(CylinderData := mpCylinderData^, bSmallSize := bSmallSize, bCalcHighPressSize := FALSE);
   // convert bar to kN
   mprMaxPressure^ := mprMaxHydrPressure^ * rCylinderSize / 10000.0;
ELSE
   mprMaxPressure^ := mprMaxHydrPressure^;
END_IF;

;#END_EDIT_BLOCK END_ALGORITHM

ALGORITHM aInit

VAR_INPUT
 pLintabOut : REFTO KAPPL_LintabData;
 prMaxPressure : REFTO REAL (* reference to calculated max. pressure *);
 prMaxHydrPressure : REFTO REAL (* reference to max. possible hydraulic pressure (depends on used pumps(s)) *);
 bUseForce : BOOL (* TRUE when using Force, FALSE when using pressure *);
 bFwd : BOOL (* TRUE if block is used for fwd movement *);
 pCylinderData : REFTO tsCylinderData (* cylinder data for calculating force only used when bUseForce is TRUE *);
END_VAR

VAR
 fbDebugTrace : FBDebugTrace;
END_VAR
#BEGIN_EDIT_BLOCK
(**************************************** WARNING ********************************************
 *** The KEBA Kemro K2 System including software is not intended for safety control tasks! ***
 ***                       For further information see Comment tab!                        ***
 *********************************************************************************************)

mbInitDone := FALSE;
mpCylinderData := pCylinderData;
mpLintabOut := pLintabOut;
mprMaxPressure := prMaxPressure;
mprMaxHydrPressure := prMaxHydrPressure;
mbFwd := bFwd;
mbUseForce := bUseForce;

IF bUseForce AND (NOT CHECK_REF(pCylinderData^)) THEN
   fbDebugTrace('pCylinderData not valid');
   RETURN;
END_IF;

IF (NOT CHECK_REF(pLintabOut^)) THEN
   fbDebugTrace('pLintabOut not valid');
   RETURN;
END_IF;

IF (NOT CHECK_REF(prMaxPressure^)) THEN
   fbDebugTrace('prMaxPressure not valid');
   RETURN;
END_IF;

IF (NOT CHECK_REF(prMaxHydrPressure^)) THEN
   fbDebugTrace('prMaxHydrPressure not valid');
   RETURN;
END_IF;

// init successful
mbInitDone := TRUE;

aCalcMaxPressure();

//update lintab
aUpdateLintabOut();

;#END_EDIT_BLOCK END_ALGORITHM

POSTUPDATE_ALGORITHM pUpdatePressure ON PU_Task_7 WITH mprMaxHydrPressure^,mpCylinderData^

#BEGIN_EDIT_BLOCK
(**************************************** WARNING ********************************************
 *** The KEBA Kemro K2 System including software is not intended for safety control tasks! ***
 ***                       For further information see Comment tab!                        ***
 *********************************************************************************************)

IF NOT mbInitDone THEN
    RETURN;
END_IF;

aCalcMaxPressure();

;#END_EDIT_BLOCK END_ALGORITHM

POSTUPDATE_ALGORITHM pUpdatePressureLintab ON PU_Task_7 WITH mprMaxHydrPressure^,mprMaxPressure^

#BEGIN_EDIT_BLOCK
(**************************************** WARNING ********************************************
 *** The KEBA Kemro K2 System including software is not intended for safety control tasks! ***
 ***                       For further information see Comment tab!                        ***
 *********************************************************************************************)

IF NOT mbInitDone THEN
    RETURN;
END_IF;

aUpdateLintabOut();

;#END_EDIT_BLOCK END_ALGORITHM

END_ALGORITHM_BLOCK

#END_OF_IEC_PART

@Puma @IecEditor 6 114 @Pou 25
@@@BEG_Comment@@@
@h    ! WARNING !
@h    The Kemro K2 system (including software) only meets category B according to EN 954-1,
@h    thus it is not intended for usage in safety-relevant control applications in the field
@h    of personal safety (e.g. emergency stop).
@h    To implement potentially necessary safety-relevant control tasks, always use additional
@h    external safety devices that are intended for the particular purpose, and meet the necessary
@h    functional safety.
@h    For further information see EN 954-1 (EN ISO 13849-1) and/or the K2-x00 user manual, chapter
@h    "CE conformity, directives and standards".
@@@END_Comment@@@

@BEG_Contents

@BEG_Func
@RT(17)FuncTreeContainer
3
@Var @RT(16)FFixCylinderData @RT(0) @T @T @DERIVED 0 @F @RT(8)FUNCTION @F
@T
@BEG_Attrib
0 @RT(0) @RT(0)
@END_Attrib
1 1 @F @F @F @F

@Var @RT(22)FCalculateCylinderSize @RT(0) @T @T @DERIVED 0 @F @RT(8)FUNCTION @F
@T
@BEG_Attrib
0 @RT(0) @RT(0)
@END_Attrib
1 1 @F @F @F @F

@Var @RT(9)CHECK_REF @RT(0) @T @T @DERIVED 0 @F @RT(23)KEBA_STANDARD_PROCEDURE @F
@T
@BEG_Attrib
0 @RT(0) @RT(0)
@END_Attrib
1 1 @F @F @F @F

@END_Func

@BEG_Const
@RT(18)ConstTreeContainer
0
@END_Const

@BEG_Export

@BEG_Kind
@ALGORITHM_BLOCK @RT(20)ABUpdateRelLintabPre @STRUCTURED_TEXT
@RT(0) @RT(0) @RT(0)
@END_Kind

@BEG_Dcl
@RT(16)DclTreeContainer
9
@Var @RT(28)sv_bCalcMaxValuesFromCylData @RT(0) @T @F @DT @RT(4)BOOL @RT(0) @T @T @BASIC 0 @F
@F @F
@T
@BEG_Attrib
3 @RT(0) @RT(117)TRUE: calculate max speed and max pressure values by using cylinder data;  FALSE: max values must be entered manually @RT(0)
@END_Attrib
1 8 @F @F @F @F

@Var @RT(9)PU_Task_7 @RT(0) @T @F @DT @RT(4)TASK @RT(0) @T @T @BASIC 0 @F
@F @F
@T
@BEG_Attrib
3 @RT(0) @RT(0) @RT(0)
@END_Attrib
1 7 @F @F @F @F

@Var @RT(11)mpLintabOut @RT(0) @T @T @REFTO 0 @F @DERIVED 0 @T @T @DT @RT(16)KAPPL_LintabData @RT(0) @T @T @UNKNOWN 0 @F
@F @F
@T
@BEG_Attrib
3 @RT(0) @RT(33)refto pressure lintab of movement @RT(0)
@END_Attrib
1 0 @F @F @F @F

@Var @RT(14)mpCylinderData @RT(0) @T @T @REFTO 0 @F @DERIVED 0 @T @T @DT @RT(14)tsCylinderData @RT(0) @T @T @UNKNOWN 0 @F
@F @F
@T
@BEG_Attrib
3 @RT(0) @RT(19)refto cylinder data @RT(0)
@END_Attrib
1 0 @F @F @F @F

@Var @RT(14)mprMaxPressure @RT(0) @T @T @REFTO 0 @T @DT @RT(4)REAL @RT(0) @T @T @BASIC 0 @F
@F @F
@T
@BEG_Attrib
3 @RT(0) @RT(49)reference to calculated max. pressure of movement @RT(0)
@END_Attrib
1 0 @F @F @F @F

@Var @RT(18)mprMaxHydrPressure @RT(0) @T @T @REFTO 0 @T @DT @RT(4)REAL @RT(0) @T @T @BASIC 0 @F
@F @F
@T
@BEG_Attrib
3 @RT(0) @RT(36)reference to max. hydraulic pressure @RT(0)
@END_Attrib
1 0 @F @F @F @F

@Var @RT(10)mbInitDone @RT(0) @T @F @DT @RT(4)BOOL @RT(0) @T @T @BASIC 0 @F
@F @F
@T
@BEG_Attrib
3 @RT(0) @RT(0) @RT(0)
@END_Attrib
1 0 @F @F @F @F

@Var @RT(10)mbUseForce @RT(0) @T @F @DT @RT(4)BOOL @RT(0) @T @T @BASIC 0 @F
@F @F
@T
@BEG_Attrib
3 @RT(0) @RT(0) @RT(0)
@END_Attrib
1 0 @F @F @F @F

@Var @RT(5)mbFwd @RT(0) @T @F @DT @RT(4)BOOL @RT(0) @T @T @BASIC 0 @F
@F @F
@T
@BEG_Attrib
3 @RT(0) @RT(0) @RT(0)
@END_Attrib
1 0 @F @F @F @F

@END_Dcl

@END_Export

@BEG_Body

5

@BEG_Export

@BEG_Algo
@ALGORITHM @RT(16)aUpdateLintabOut @STRUCTURED_TEXT
@RT(0) @RT(0) @RT(0) @F @F
@END_Algo

@BEG_Dcl
@RT(16)DclTreeContainer
0
@END_Dcl

@END_Export

@BEG_Export

@BEG_Algo
@ALGORITHM @RT(16)aCalcMaxPressure @STRUCTURED_TEXT
@RT(0) @RT(0) @RT(0) @F @F
@END_Algo

@BEG_Dcl
@RT(16)DclTreeContainer
3
@Var @RT(13)rCylinderSize @RT(0) @T @F @DT @RT(4)REAL @RT(0) @T @T @BASIC 0 @F
@F @F
@T
@BEG_Attrib
3 @RT(0) @RT(23)size of cylinder im mm˛ @RT(0)
@END_Attrib
1 4 @F @F @F @F

@Var @RT(3)tmp @RT(0) @T @F @DT @RT(4)BOOL @RT(0) @T @T @BASIC 0 @F
@F @F
@T
@BEG_Attrib
3 @RT(0) @RT(0) @RT(0)
@END_Attrib
1 4 @F @F @F @F

@Var @RT(10)bSmallSize @RT(0) @T @F @DT @RT(4)BOOL @RT(0) @T @T @BASIC 0 @F
@F @F
@T
@BEG_Attrib
3 @RT(0) @RT(0) @RT(0)
@END_Attrib
1 0 @F @F @F @F

@END_Dcl

@END_Export

@BEG_Export

@BEG_Algo
@ALGORITHM @RT(5)aInit @STRUCTURED_TEXT
@RT(0) @RT(0) @RT(0) @F @F
@END_Algo

@BEG_Dcl
@RT(16)DclTreeContainer
7
@Var @RT(10)pLintabOut @RT(0) @T @T @REFTO 0 @F @DERIVED 0 @T @T @DT @RT(16)KAPPL_LintabData @RT(0) @T @T @UNKNOWN 0 @F
@F @F
@T
@BEG_Attrib
3 @RT(0) @RT(0) @RT(0)
@END_Attrib
1 1 @F @F @F @F

@Var @RT(13)prMaxPressure @RT(0) @T @T @REFTO 0 @T @DT @RT(4)REAL @RT(0) @T @T @BASIC 0 @F
@F @F
@T
@BEG_Attrib
3 @RT(0) @RT(37)reference to calculated max. pressure @RT(0)
@END_Attrib
1 1 @F @F @F @F

@Var @RT(17)prMaxHydrPressure @RT(0) @T @T @REFTO 0 @T @DT @RT(4)REAL @RT(0) @T @T @BASIC 0 @F
@F @F
@T
@BEG_Attrib
3 @RT(0) @RT(72)reference to max. possible hydraulic pressure (depends on used pumps(s)) @RT(0)
@END_Attrib
1 1 @F @F @F @F

@Var @RT(9)bUseForce @RT(0) @T @F @DT @RT(4)BOOL @RT(0) @T @T @BASIC 0 @F
@F @F
@T
@BEG_Attrib
3 @RT(0) @RT(48)TRUE when using Force, FALSE when using pressure @RT(0)
@END_Attrib
1 1 @F @F @F @F

@Var @RT(4)bFwd @RT(0) @T @F @DT @RT(4)BOOL @RT(0) @T @T @BASIC 0 @F
@F @F
@T
@BEG_Attrib
3 @RT(0) @RT(38)TRUE if block is used for fwd movement @RT(0)
@END_Attrib
1 1 @F @F @F @F

@Var @RT(13)pCylinderData @RT(0) @T @T @REFTO 0 @F @DERIVED 0 @T @T @DT @RT(14)tsCylinderData @RT(0) @T @T @UNKNOWN 0 @F
@F @F
@T
@BEG_Attrib
3 @RT(0) @RT(68)cylinder data for calculating force only used when bUseForce is TRUE @RT(0)
@END_Attrib
1 1 @F @F @F @F

@Var @RT(12)fbDebugTrace @RT(0) @T @T @DERIVED 0 @T @T @DT @RT(12)FBDebugTrace @RT(0) @T @T @UNKNOWN 0 @F
@F @F
@T
@BEG_Attrib
3 @RT(0) @RT(0) @RT(0)
@END_Attrib
1 0 @F @F @F @F

@END_Dcl

@END_Export

@BEG_Export

@BEG_Algo
@POSTUPDATE_ALGORITHM @RT(15)pUpdatePressure @STRUCTURED_TEXT
@RT(0) @RT(35)mprMaxHydrPressure^,mpCylinderData^ @RT(9)PU_Task_7 @F @F
@END_Algo

@BEG_Dcl
@RT(16)DclTreeContainer
0
@END_Dcl

@END_Export

@BEG_Export

@BEG_Algo
@POSTUPDATE_ALGORITHM @RT(21)pUpdatePressureLintab @STRUCTURED_TEXT
@RT(0) @RT(35)mprMaxHydrPressure^,mprMaxPressure^ @RT(9)PU_Task_7 @F @F
@END_Algo

@BEG_Dcl
@RT(16)DclTreeContainer
0
@END_Dcl

@END_Export

@BEG_Body
@TL(13)
(**************************************** WARNING ********************************************
 *** The KEBA Kemro K2 System including software is not intended for safety control tasks! ***
 ***                       For further information see Comment tab!                        ***
 *********************************************************************************************)

// save data to Pre lintab
// normally a 1:1 lintab
mpLintabOut^.LintabPoints.uNoOfPoints := 2;
mpLintabOut^.LintabPoints.Point[1].rX := 0.0;
mpLintabOut^.LintabPoints.Point[1].rY := 0.0;
mpLintabOut^.LintabPoints.Point[2].rX := mprMaxPressure^;
mpLintabOut^.LintabPoints.Point[2].rY := mprMaxHydrPressure^;

@END_Body

@@@BEG_Comment@@@
@TL(0)

@@@END_Comment@@@

@BEG_Body
@TL(21)
(**************************************** WARNING ********************************************
 *** The KEBA Kemro K2 System including software is not intended for safety control tasks! ***
 ***                       For further information see Comment tab!                        ***
 *********************************************************************************************)

IF NOT sv_bCalcMaxValuesFromCylData THEN
   // no calculation necessary
   RETURN;
END_IF;

IF mbUseForce THEN
   tmp := FFixCylinderData(mpCylinderData);
   bSmallSize := mbFwd AND mpCylinderData^.bUseSmallSize OR
                 ((NOT mbFwd AND NOT mpCylinderData^.bUseSmallSize));
   rCylinderSize := FCalculateCylinderSize(CylinderData := mpCylinderData^, bSmallSize := bSmallSize, bCalcHighPressSize := FALSE);
   // convert bar to kN
   mprMaxPressure^ := mprMaxHydrPressure^ * rCylinderSize / 10000.0;
ELSE
   mprMaxPressure^ := mprMaxHydrPressure^;
END_IF;

@END_Body

@@@BEG_Comment@@@
@TL(0)

@@@END_Comment@@@

@BEG_Body
@TL(41)
(**************************************** WARNING ********************************************
 *** The KEBA Kemro K2 System including software is not intended for safety control tasks! ***
 ***                       For further information see Comment tab!                        ***
 *********************************************************************************************)

mbInitDone := FALSE;
mpCylinderData := pCylinderData;
mpLintabOut := pLintabOut;
mprMaxPressure := prMaxPressure;
mprMaxHydrPressure := prMaxHydrPressure;
mbFwd := bFwd;
mbUseForce := bUseForce;

IF bUseForce AND (NOT CHECK_REF(pCylinderData^)) THEN
   fbDebugTrace('pCylinderData not valid');
   RETURN;
END_IF;

IF (NOT CHECK_REF(pLintabOut^)) THEN
   fbDebugTrace('pLintabOut not valid');
   RETURN;
END_IF;

IF (NOT CHECK_REF(prMaxPressure^)) THEN
   fbDebugTrace('prMaxPressure not valid');
   RETURN;
END_IF;

IF (NOT CHECK_REF(prMaxHydrPressure^)) THEN
   fbDebugTrace('prMaxHydrPressure not valid');
   RETURN;
END_IF;

// init successful
mbInitDone := TRUE;

aCalcMaxPressure();

//update lintab
aUpdateLintabOut();

@END_Body

@@@BEG_Comment@@@
@TL(0)

@@@END_Comment@@@

@BEG_Body
@TL(11)
(**************************************** WARNING ********************************************
 *** The KEBA Kemro K2 System including software is not intended for safety control tasks! ***
 ***                       For further information see Comment tab!                        ***
 *********************************************************************************************)

IF NOT mbInitDone THEN
    RETURN;
END_IF;

aCalcMaxPressure();

@END_Body

@@@BEG_Comment@@@
@TL(0)

@@@END_Comment@@@

@BEG_Body
@TL(11)
(**************************************** WARNING ********************************************
 *** The KEBA Kemro K2 System including software is not intended for safety control tasks! ***
 ***                       For further information see Comment tab!                        ***
 *********************************************************************************************)

IF NOT mbInitDone THEN
    RETURN;
END_IF;

aUpdateLintabOut();

@END_Body

@@@BEG_Comment@@@
@TL(0)

@@@END_Comment@@@
@END_Body

@END_Contents
